   DATA[2227,0] := 2.649009;
   DATA[2227,1] := 864.9738;
   DATA[2227,2] := 2.0;
   DATA[2227,3] := 2.0;
   DATA[2227,4] := 262.3366;
   DATA[2227,5] := 8.394514;
   DATA[2227,6] := 330.2999;
   DATA[2227,7] := 2.461539;
   DATA[2227,8] := 2.0;
   DATA[2227,9] := 2.0;
   DATA[2227,10] := 2.0;
   DATA[2227,11] := 19.73878;
   DATA[2227,12] := 2.209653;
   DATA[2227,13] := 811.05;
   DATA[2227,14] := 1.0;
   DATA[2227,15] := 2.0;
   DATA[2227,16] := 1.0;
   DATA[2227,17] := 1.0;
   DATA[2227,18] := 1.0;
   DATA[2227,19] := 2.0;
   DATA[2227,20] := 148.808;
   DATA[2227,21] := 155.0884;
   DATA[2227,22] := 1.715567;
   DATA[2227,23] := 847.5134;
   DATA[2227,24] := 2.0;
   DATA[2227,25] := 2.0;
   DATA[2227,26] := 7.873815;
   DATA[2227,27] := 144.2194;
   DATA[2227,28] := 261.8559;
   DATA[2227,29] := 11.88157;
   DATA[2227,30] := 1.726865;
   DATA[2227,31] := 1.281927;
   DATA[2227,32] := 0.7352687;
   DATA[2227,33] := 0.3084905;
   DATA[2227,34] := 2.0;
   DATA[2227,35] := 250.016;
   DATA[2227,36] := 1.69801;
   DATA[2227,37] := 188.9259;
   DATA[2227,38] := 0.000128152;
   DATA[2227,39] := 1.0;
   DATA[2227,40] := 1.0;
   DATA[2228,0] := 2.653813;
   DATA[2228,1] := 865.013;
   DATA[2228,2] := 2.0;
   DATA[2228,3] := 2.0;
   DATA[2228,4] := 262.3366;
   DATA[2228,5] := 8.394514;
   DATA[2228,6] := 330.2999;
   DATA[2228,7] := 2.461539;
   DATA[2228,8] := 2.0;
   DATA[2228,9] := 2.0;
   DATA[2228,10] := 2.0;
   DATA[2228,11] := 19.73878;
   DATA[2228,12] := 2.209653;
   DATA[2228,13] := 811.01;
   DATA[2228,14] := 1.0;
   DATA[2228,15] := 2.0;
   DATA[2228,16] := 1.0;
   DATA[2228,17] := 1.0;
   DATA[2228,18] := 1.0;
   DATA[2228,19] := 2.0;
   DATA[2228,20] := 148.808;
   DATA[2228,21] := 155.0884;
   DATA[2228,22] := 1.715567;
   DATA[2228,23] := 847.5903;
   DATA[2228,24] := 2.0;
   DATA[2228,25] := 2.0;
   DATA[2228,26] := 7.873815;
   DATA[2228,27] := 144.2194;
   DATA[2228,28] := 261.8559;
   DATA[2228,29] := 11.88157;
   DATA[2228,30] := 1.726865;
   DATA[2228,31] := 1.281927;
   DATA[2228,32] := 0.7352687;
   DATA[2228,33] := 0.3084905;
   DATA[2228,34] := 2.0;
   DATA[2228,35] := 249.9359;
   DATA[2228,36] := 1.69801;
   DATA[2228,37] := 188.9259;
   DATA[2228,38] := 0.000128152;
   DATA[2228,39] := 1.0;
   DATA[2228,40] := 1.0;
   DATA[2229,0] := 2.643564;
   DATA[2229,1] := 864.8168;
   DATA[2229,2] := 2.0;
   DATA[2229,3] := 2.0;
   DATA[2229,4] := 262.3366;
   DATA[2229,5] := 8.394514;
   DATA[2229,6] := 330.2999;
   DATA[2229,7] := 2.460129;
   DATA[2229,8] := 2.0;
   DATA[2229,9] := 2.0;
   DATA[2229,10] := 2.0;
   DATA[2229,11] := 19.82201;
   DATA[2229,12] := 2.207603;
   DATA[2229,13] := 811.01;
   DATA[2229,14] := 1.0;
   DATA[2229,15] := 2.0;
   DATA[2229,16] := 1.0;
   DATA[2229,17] := 1.0;
   DATA[2229,18] := 1.0;
   DATA[2229,19] := 2.0;
   DATA[2229,20] := 148.808;
   DATA[2229,21] := 155.0884;
   DATA[2229,22] := 1.716849;
   DATA[2229,23] := 847.6288;
   DATA[2229,24] := 2.0;
   DATA[2229,25] := 2.0;
   DATA[2229,26] := 7.873815;
   DATA[2229,27] := 144.2194;
   DATA[2229,28] := 261.8559;
   DATA[2229,29] := 12.11228;
   DATA[2229,30] := 1.726865;
   DATA[2229,31] := 1.281927;
   DATA[2229,32] := 0.7352687;
   DATA[2229,33] := 0.3084905;
   DATA[2229,34] := 2.0;
   DATA[2229,35] := 249.9359;
   DATA[2229,36] := 1.69801;
   DATA[2229,37] := 188.9259;
   DATA[2229,38] := 0.000128152;
   DATA[2229,39] := 1.0;
   DATA[2229,40] := 1.0;
   DATA[2230,0] := 2.624988;
   DATA[2230,1] := 864.9738;
   DATA[2230,2] := 2.0;
   DATA[2230,3] := 2.0;
   DATA[2230,4] := 262.3366;
   DATA[2230,5] := 8.394514;
   DATA[2230,6] := 330.2999;
   DATA[2230,7] := 2.458206;
   DATA[2230,8] := 2.0;
   DATA[2230,9] := 2.0;
   DATA[2230,10] := 2.0;
   DATA[2230,11] := 19.82201;
   DATA[2230,12] := 2.207347;
   DATA[2230,13] := 810.9299;
   DATA[2230,14] := 1.0;
   DATA[2230,15] := 2.0;
   DATA[2230,16] := 1.0;
   DATA[2230,17] := 1.0;
   DATA[2230,18] := 1.0;
   DATA[2230,19] := 2.0;
   DATA[2230,20] := 148.808;
   DATA[2230,21] := 155.0884;
   DATA[2230,22] := 1.717361;
   DATA[2230,23] := 847.7057;
   DATA[2230,24] := 2.0;
   DATA[2230,25] := 2.0;
   DATA[2230,26] := 7.873815;
   DATA[2230,27] := 144.2194;
   DATA[2230,28] := 261.8559;
   DATA[2230,29] := 12.11228;
   DATA[2230,30] := 1.726865;
   DATA[2230,31] := 1.281927;
   DATA[2230,32] := 0.7352687;
   DATA[2230,33] := 0.3084905;
   DATA[2230,34] := 2.0;
   DATA[2230,35] := 249.9359;
   DATA[2230,36] := 1.69801;
   DATA[2230,37] := 188.9259;
   DATA[2230,38] := 0.000128152;
   DATA[2230,39] := 1.0;
   DATA[2230,40] := 1.0;
   DATA[2231,0] := 2.620504;
   DATA[2231,1] := 865.013;
   DATA[2231,2] := 2.0;
   DATA[2231,3] := 2.0;
   DATA[2231,4] := 262.3366;
   DATA[2231,5] := 8.394514;
   DATA[2231,6] := 330.2999;
   DATA[2231,7] := 2.458078;
   DATA[2231,8] := 2.0;
   DATA[2231,9] := 2.0;
   DATA[2231,10] := 2.0;
   DATA[2231,11] := 19.82201;
   DATA[2231,12] := 2.207347;
   DATA[2231,13] := 810.8498;
   DATA[2231,14] := 1.0;
   DATA[2231,15] := 2.0;
   DATA[2231,16] := 1.0;
   DATA[2231,17] := 1.0;
   DATA[2231,18] := 1.0;
   DATA[2231,19] := 2.0;
   DATA[2231,20] := 148.808;
   DATA[2231,21] := 155.0884;
   DATA[2231,22] := 1.717361;
   DATA[2231,23] := 847.821;
   DATA[2231,24] := 2.0;
   DATA[2231,25] := 2.0;
   DATA[2231,26] := 7.873815;
   DATA[2231,27] := 144.2194;
   DATA[2231,28] := 261.8559;
   DATA[2231,29] := 12.11228;
   DATA[2231,30] := 1.728531;
   DATA[2231,31] := 1.281927;
   DATA[2231,32] := 0.7352687;
   DATA[2231,33] := 0.3084905;
   DATA[2231,34] := 2.0;
   DATA[2231,35] := 249.9359;
   DATA[2231,36] := 1.69801;
   DATA[2231,37] := 188.9259;
   DATA[2231,38] := 0.000128152;
   DATA[2231,39] := 1.0;
   DATA[2231,40] := 1.0;
   DATA[2232,0] := 2.616981;
   DATA[2232,1] := 865.013;
   DATA[2232,2] := 2.0;
   DATA[2232,3] := 2.0;
   DATA[2232,4] := 262.3366;
   DATA[2232,5] := 8.394514;
   DATA[2232,6] := 330.2999;
   DATA[2232,7] := 2.455772;
   DATA[2232,8] := 2.0;
   DATA[2232,9] := 2.0;
   DATA[2232,10] := 2.0;
   DATA[2232,11] := 19.74198;
   DATA[2232,12] := 2.207347;
   DATA[2232,13] := 811.1302;
   DATA[2232,14] := 1.0;
   DATA[2232,15] := 2.0;
   DATA[2232,16] := 1.0;
   DATA[2232,17] := 1.0;
   DATA[2232,18] := 1.0;
   DATA[2232,19] := 2.0;
   DATA[2232,20] := 148.808;
   DATA[2232,21] := 155.0884;
   DATA[2232,22] := 1.717361;
   DATA[2232,23] := 847.6288;
   DATA[2232,24] := 2.0;
   DATA[2232,25] := 2.0;
   DATA[2232,26] := 7.873815;
   DATA[2232,27] := 144.2194;
   DATA[2232,28] := 261.8559;
   DATA[2232,29] := 12.11228;
   DATA[2232,30] := 1.728659;
   DATA[2232,31] := 1.268989;
   DATA[2232,32] := 0.7352687;
   DATA[2232,33] := 0.3084905;
   DATA[2232,34] := 2.0;
   DATA[2232,35] := 250.1122;
   DATA[2232,36] := 1.69801;
   DATA[2232,37] := 188.9259;
   DATA[2232,38] := 0.000128152;
   DATA[2232,39] := 1.0;
   DATA[2232,40] := 1.0;
   DATA[2233,0] := 2.609615;
   DATA[2233,1] := 865.2485;
   DATA[2233,2] := 2.0;
   DATA[2233,3] := 2.0;
   DATA[2233,4] := 262.3366;
   DATA[2233,5] := 8.396757;
   DATA[2233,6] := 330.2999;
   DATA[2233,7] := 2.456412;
   DATA[2233,8] := 2.0;
   DATA[2233,9] := 2.0;
   DATA[2233,10] := 2.0;
   DATA[2233,11] := 19.71957;
   DATA[2233,12] := 2.207347;
   DATA[2233,13] := 811.1302;
   DATA[2233,14] := 1.0;
   DATA[2233,15] := 2.0;
   DATA[2233,16] := 1.0;
   DATA[2233,17] := 1.0;
   DATA[2233,18] := 1.0;
   DATA[2233,19] := 2.0;
   DATA[2233,20] := 148.808;
   DATA[2233,21] := 155.0884;
   DATA[2233,22] := 1.717361;
   DATA[2233,23] := 847.821;
   DATA[2233,24] := 2.0;
   DATA[2233,25] := 2.0;
   DATA[2233,26] := 7.873815;
   DATA[2233,27] := 144.2194;
   DATA[2233,28] := 261.8559;
   DATA[2233,29] := 12.11228;
   DATA[2233,30] := 1.728659;
   DATA[2233,31] := 1.261816;
   DATA[2233,32] := 0.7352687;
   DATA[2233,33] := 0.3084905;
   DATA[2233,34] := 2.0;
   DATA[2233,35] := 250.2243;
   DATA[2233,36] := 1.69801;
   DATA[2233,37] := 188.9259;
   DATA[2233,38] := 0.000128152;
   DATA[2233,39] := 1.0;
   DATA[2233,40] := 1.0;
   DATA[2234,0] := 2.588156;
   DATA[2234,1] := 865.013;
   DATA[2234,2] := 2.0;
   DATA[2234,3] := 2.0;
   DATA[2234,4] := 262.3366;
   DATA[2234,5] := 8.396757;
   DATA[2234,6] := 330.2999;
   DATA[2234,7] := 2.458078;
   DATA[2234,8] := 2.0;
   DATA[2234,9] := 2.0;
   DATA[2234,10] := 2.0;
   DATA[2234,11] := 19.71957;
   DATA[2234,12] := 2.206963;
   DATA[2234,13] := 811.05;
   DATA[2234,14] := 1.0;
   DATA[2234,15] := 2.0;
   DATA[2234,16] := 1.0;
   DATA[2234,17] := 1.0;
   DATA[2234,18] := 1.0;
   DATA[2234,19] := 2.0;
   DATA[2234,20] := 148.808;
   DATA[2234,21] := 155.0884;
   DATA[2234,22] := 1.717361;
   DATA[2234,23] := 847.8979;
   DATA[2234,24] := 2.0;
   DATA[2234,25] := 2.0;
   DATA[2234,26] := 7.873815;
   DATA[2234,27] := 144.2194;
   DATA[2234,28] := 261.8559;
   DATA[2234,29] := 11.88157;
   DATA[2234,30] := 1.728659;
   DATA[2234,31] := 1.261816;
   DATA[2234,32] := 0.7352687;
   DATA[2234,33] := 0.3082983;
   DATA[2234,34] := 2.0;
   DATA[2234,35] := 250.2243;
   DATA[2234,36] := 1.69801;
   DATA[2234,37] := 188.974;
   DATA[2234,38] := 0.000128152;
   DATA[2234,39] := 1.0;
   DATA[2234,40] := 1.0;
   DATA[2235,0] := 2.5699;
   DATA[2235,1] := 864.9345;
   DATA[2235,2] := 2.0;
   DATA[2235,3] := 2.0;
   DATA[2235,4] := 262.3366;
   DATA[2235,5] := 8.396757;
   DATA[2235,6] := 330.2999;
   DATA[2235,7] := 2.458078;
   DATA[2235,8] := 2.0;
   DATA[2235,9] := 2.0;
   DATA[2235,10] := 2.0;
   DATA[2235,11] := 19.71957;
   DATA[2235,12] := 2.206963;
   DATA[2235,13] := 811.01;
   DATA[2235,14] := 1.0;
   DATA[2235,15] := 2.0;
   DATA[2235,16] := 1.0;
   DATA[2235,17] := 1.0;
   DATA[2235,18] := 1.0;
   DATA[2235,19] := 2.0;
   DATA[2235,20] := 148.808;
   DATA[2235,21] := 155.0372;
   DATA[2235,22] := 1.717361;
   DATA[2235,23] := 847.9364;
   DATA[2235,24] := 2.0;
   DATA[2235,25] := 2.0;
   DATA[2235,26] := 7.873815;
   DATA[2235,27] := 144.2194;
   DATA[2235,28] := 261.8559;
   DATA[2235,29] := 11.88157;
   DATA[2235,30] := 1.728659;
   DATA[2235,31] := 1.276419;
   DATA[2235,32] := 0.7352687;
   DATA[2235,33] := 0.3074016;
   DATA[2235,34] := 2.0;
   DATA[2235,35] := 250.2243;
   DATA[2235,36] := 1.69801;
   DATA[2235,37] := 189.1182;
   DATA[2235,38] := 0.000128152;
   DATA[2235,39] := 1.0;
   DATA[2235,40] := 1.0;
   DATA[2236,0] := 2.554847;
   DATA[2236,1] := 864.8168;
   DATA[2236,2] := 2.0;
   DATA[2236,3] := 2.0;
   DATA[2236,4] := 262.3366;
   DATA[2236,5] := 8.396757;
   DATA[2236,6] := 330.2999;
   DATA[2236,7] := 2.458078;
   DATA[2236,8] := 2.0;
   DATA[2236,9] := 2.0;
   DATA[2236,10] := 2.0;
   DATA[2236,11] := 19.71957;
   DATA[2236,12] := 2.206963;
   DATA[2236,13] := 811.05;
   DATA[2236,14] := 1.0;
   DATA[2236,15] := 2.0;
   DATA[2236,16] := 1.0;
   DATA[2236,17] := 1.0;
   DATA[2236,18] := 1.0;
   DATA[2236,19] := 2.0;
   DATA[2236,20] := 148.808;
   DATA[2236,21] := 155.0372;
   DATA[2236,22] := 1.718771;
   DATA[2236,23] := 847.821;
   DATA[2236,24] := 2.0;
   DATA[2236,25] := 2.0;
   DATA[2236,26] := 7.873815;
   DATA[2236,27] := 144.2194;
   DATA[2236,28] := 261.8559;
   DATA[2236,29] := 11.88157;
   DATA[2236,30] := 1.728659;
   DATA[2236,31] := 1.282311;
   DATA[2236,32] := 0.7352687;
   DATA[2236,33] := 0.306761;
   DATA[2236,34] := 2.0;
   DATA[2236,35] := 250.3365;
   DATA[2236,36] := 1.69801;
   DATA[2236,37] := 189.1182;
   DATA[2236,38] := 0.000128152;
   DATA[2236,39] := 1.0;
   DATA[2236,40] := 1.0;
   DATA[2237,0] := 2.53467;
   DATA[2237,1] := 864.4243;
   DATA[2237,2] := 2.0;
   DATA[2237,3] := 2.0;
   DATA[2237,4] := 262.3366;
   DATA[2237,5] := 8.396757;
   DATA[2237,6] := 330.2999;
   DATA[2237,7] := 2.457438;
   DATA[2237,8] := 2.0;
   DATA[2237,9] := 2.0;
   DATA[2237,10] := 2.0;
   DATA[2237,11] := 19.72598;
   DATA[2237,12] := 2.209653;
   DATA[2237,13] := 810.6495;
   DATA[2237,14] := 1.0;
   DATA[2237,15] := 2.0;
   DATA[2237,16] := 1.0;
   DATA[2237,17] := 1.0;
   DATA[2237,18] := 1.0;
   DATA[2237,19] := 2.0;
   DATA[2237,20] := 148.808;
   DATA[2237,21] := 155.0372;
   DATA[2237,22] := 1.718771;
   DATA[2237,23] := 847.9364;
   DATA[2237,24] := 2.0;
   DATA[2237,25] := 2.0;
   DATA[2237,26] := 7.873815;
   DATA[2237,27] := 144.2194;
   DATA[2237,28] := 261.8559;
   DATA[2237,29] := 11.88157;
   DATA[2237,30] := 1.728659;
   DATA[2237,31] := 1.26758;
   DATA[2237,32] := 0.7352687;
   DATA[2237,33] := 0.306761;
   DATA[2237,34] := 2.0;
   DATA[2237,35] := 250.3365;
   DATA[2237,36] := 1.69801;
   DATA[2237,37] := 189.1182;
   DATA[2237,38] := 0.000128152;
   DATA[2237,39] := 1.0;
   DATA[2237,40] := 1.0;
   DATA[2238,0] := 2.516734;
   DATA[2238,1] := 864.1887;
   DATA[2238,2] := 2.0;
   DATA[2238,3] := 2.0;
   DATA[2238,4] := 262.3366;
   DATA[2238,5] := 8.396757;
   DATA[2238,6] := 330.2999;
   DATA[2238,7] := 2.456541;
   DATA[2238,8] := 2.0;
   DATA[2238,9] := 2.0;
   DATA[2238,10] := 2.0;
   DATA[2238,11] := 19.72598;
   DATA[2238,12] := 2.209653;
   DATA[2238,13] := 810.8498;
   DATA[2238,14] := 1.0;
   DATA[2238,15] := 2.0;
   DATA[2238,16] := 1.0;
   DATA[2238,17] := 1.0;
   DATA[2238,18] := 1.0;
   DATA[2238,19] := 2.0;
   DATA[2238,20] := 148.808;
   DATA[2238,21] := 155.0372;
   DATA[2238,22] := 1.718771;
   DATA[2238,23] := 848.2056;
   DATA[2238,24] := 2.0;
   DATA[2238,25] := 2.0;
   DATA[2238,26] := 7.873815;
   DATA[2238,27] := 144.2194;
   DATA[2238,28] := 261.8559;
   DATA[2238,29] := 11.88157;
   DATA[2238,30] := 1.727378;
   DATA[2238,31] := 1.256821;
   DATA[2238,32] := 0.7352687;
   DATA[2238,33] := 0.306761;
   DATA[2238,34] := 2.0;
   DATA[2238,35] := 250.4646;
   DATA[2238,36] := 1.69801;
   DATA[2238,37] := 189.1182;
   DATA[2238,38] := 0.000128152;
   DATA[2238,39] := 1.0;
   DATA[2238,40] := 1.0;
   DATA[2239,0] := 2.498479;
   DATA[2239,1] := 864.3457;
   DATA[2239,2] := 2.0;
   DATA[2239,3] := 2.0;
   DATA[2239,4] := 262.3366;
   DATA[2239,5] := 8.394835;
   DATA[2239,6] := 330.2999;
   DATA[2239,7] := 2.456541;
   DATA[2239,8] := 2.0;
   DATA[2239,9] := 2.0;
   DATA[2239,10] := 2.0;
   DATA[2239,11] := 19.75799;
   DATA[2239,12] := 2.208244;
   DATA[2239,13] := 810.5694;
   DATA[2239,14] := 1.0;
   DATA[2239,15] := 2.0;
   DATA[2239,16] := 1.0;
   DATA[2239,17] := 1.0;
   DATA[2239,18] := 1.0;
   DATA[2239,19] := 2.0;
   DATA[2239,20] := 148.808;
   DATA[2239,21] := 155.0372;
   DATA[2239,22] := 1.718771;
   DATA[2239,23] := 848.1671;
   DATA[2239,24] := 2.0;
   DATA[2239,25] := 2.0;
   DATA[2239,26] := 7.873815;
   DATA[2239,27] := 144.2194;
   DATA[2239,28] := 261.8559;
   DATA[2239,29] := 12.03538;
   DATA[2239,30] := 1.725968;
   DATA[2239,31] := 1.254259;
   DATA[2239,32] := 0.7352687;
   DATA[2239,33] := 0.306761;
   DATA[2239,34] := 2.0;
   DATA[2239,35] := 250.4646;
   DATA[2239,36] := 1.69801;
   DATA[2239,37] := 189.1182;
   DATA[2239,38] := 0.000128152;
   DATA[2239,39] := 1.0;
   DATA[2239,40] := 1.0;
   DATA[2240,0] := 2.484707;
   DATA[2240,1] := 863.9532;
   DATA[2240,2] := 2.0;
   DATA[2240,3] := 2.0;
   DATA[2240,4] := 262.3366;
   DATA[2240,5] := 8.394835;
   DATA[2240,6] := 330.2999;
   DATA[2240,7] := 2.456541;
   DATA[2240,8] := 2.0;
   DATA[2240,9] := 2.0;
   DATA[2240,10] := 2.0;
   DATA[2240,11] := 19.75799;
   DATA[2240,12] := 2.20645;
   DATA[2240,13] := 810.5294;
   DATA[2240,14] := 1.0;
   DATA[2240,15] := 2.0;
   DATA[2240,16] := 1.0;
   DATA[2240,17] := 1.0;
   DATA[2240,18] := 1.0;
   DATA[2240,19] := 2.0;
   DATA[2240,20] := 148.808;
   DATA[2240,21] := 155.0884;
   DATA[2240,22] := 1.717874;
   DATA[2240,23] := 848.3209;
   DATA[2240,24] := 2.0;
   DATA[2240,25] := 2.0;
   DATA[2240,26] := 7.873815;
   DATA[2240,27] := 144.2194;
   DATA[2240,28] := 261.7278;
   DATA[2240,29] := 12.15073;
   DATA[2240,30] := 1.724686;
   DATA[2240,31] := 1.254259;
   DATA[2240,32] := 0.7352687;
   DATA[2240,33] := 0.306761;
   DATA[2240,34] := 2.0;
   DATA[2240,35] := 250.4646;
   DATA[2240,36] := 1.69801;
   DATA[2240,37] := 189.1182;
   DATA[2240,38] := 0.000128152;
   DATA[2240,39] := 1.0;
   DATA[2240,40] := 1.0;
   DATA[2241,0] := 2.472216;
   DATA[2241,1] := 863.2859;
   DATA[2241,2] := 2.0;
   DATA[2241,3] := 2.0;
   DATA[2241,4] := 262.3366;
   DATA[2241,5] := 8.394835;
   DATA[2241,6] := 330.2999;
   DATA[2241,7] := 2.455643;
   DATA[2241,8] := 2.0;
   DATA[2241,9] := 2.0;
   DATA[2241,10] := 2.0;
   DATA[2241,11] := 19.73238;
   DATA[2241,12] := 2.20645;
   DATA[2241,13] := 810.4493;
   DATA[2241,14] := 1.0;
   DATA[2241,15] := 2.0;
   DATA[2241,16] := 1.0;
   DATA[2241,17] := 1.0;
   DATA[2241,18] := 1.0;
   DATA[2241,19] := 2.0;
   DATA[2241,20] := 148.808;
   DATA[2241,21] := 155.191;
   DATA[2241,22] := 1.717489;
   DATA[2241,23] := 848.3978;
   DATA[2241,24] := 2.0;
   DATA[2241,25] := 2.0;
   DATA[2241,26] := 7.873815;
   DATA[2241,27] := 144.2194;
   DATA[2241,28] := 261.7278;
   DATA[2241,29] := 12.15073;
   DATA[2241,30] := 1.724686;
   DATA[2241,31] := 1.270783;
   DATA[2241,32] := 0.7352687;
   DATA[2241,33] := 0.306761;
   DATA[2241,34] := 2.0;
   DATA[2241,35] := 250.3365;
   DATA[2241,36] := 1.69801;
   DATA[2241,37] := 189.1182;
   DATA[2241,38] := 0.000128152;
   DATA[2241,39] := 1.0;
   DATA[2241,40] := 1.0;
   DATA[2242,0] := 2.460366;
   DATA[2242,1] := 863.0897;
   DATA[2242,2] := 2.0;
   DATA[2242,3] := 2.0;
   DATA[2242,4] := 262.3366;
   DATA[2242,5] := 8.394835;
   DATA[2242,6] := 330.2999;
   DATA[2242,7] := 2.455643;
   DATA[2242,8] := 2.0;
   DATA[2242,9] := 2.0;
   DATA[2242,10] := 2.0;
   DATA[2242,11] := 19.70037;
   DATA[2242,12] := 2.20645;
   DATA[2242,13] := 810.249;
   DATA[2242,14] := 1.0;
   DATA[2242,15] := 2.0;
   DATA[2242,16] := 1.0;
   DATA[2242,17] := 1.0;
   DATA[2242,18] := 1.0;
   DATA[2242,19] := 2.0;
   DATA[2242,20] := 148.808;
   DATA[2242,21] := 155.191;
   DATA[2242,22] := 1.717489;
   DATA[2242,23] := 848.5516;
   DATA[2242,24] := 2.0;
   DATA[2242,25] := 2.0;
   DATA[2242,26] := 7.873815;
   DATA[2242,27] := 144.2451;
   DATA[2242,28] := 261.7278;
   DATA[2242,29] := 12.15073;
   DATA[2242,30] := 1.724686;
   DATA[2242,31] := 1.272064;
   DATA[2242,32] := 0.7352687;
   DATA[2242,33] := 0.3075297;
   DATA[2242,34] := 2.0;
   DATA[2242,35] := 250.2403;
   DATA[2242,36] := 1.69801;
   DATA[2242,37] := 189.1182;
   DATA[2242,38] := 0.000128152;
   DATA[2242,39] := 1.0;
   DATA[2242,40] := 1.0;
   DATA[2243,0] := 2.445633;
   DATA[2243,1] := 863.0897;
   DATA[2243,2] := 2.0;
   DATA[2243,3] := 2.0;
   DATA[2243,4] := 262.3366;
   DATA[2243,5] := 8.394835;
   DATA[2243,6] := 330.2999;
   DATA[2243,7] := 2.455643;
   DATA[2243,8] := 2.0;
   DATA[2243,9] := 2.0;
   DATA[2243,10] := 2.0;
   DATA[2243,11] := 19.70037;
   DATA[2243,12] := 2.20645;
   DATA[2243,13] := 810.3291;
   DATA[2243,14] := 1.0;
   DATA[2243,15] := 2.0;
   DATA[2243,16] := 1.0;
   DATA[2243,17] := 1.0;
   DATA[2243,18] := 1.0;
   DATA[2243,19] := 2.0;
   DATA[2243,20] := 148.808;
   DATA[2243,21] := 155.191;
   DATA[2243,22] := 1.717489;
   DATA[2243,23] := 847.9364;
   DATA[2243,24] := 2.0;
   DATA[2243,25] := 2.0;
   DATA[2243,26] := 7.873815;
   DATA[2243,27] := 144.2451;
   DATA[2243,28] := 261.7278;
   DATA[2243,29] := 12.15073;
   DATA[2243,30] := 1.724686;
   DATA[2243,31] := 1.272064;
   DATA[2243,32] := 0.7352687;
   DATA[2243,33] := 0.3079781;
   DATA[2243,34] := 2.0;
   DATA[2243,35] := 250.2403;
   DATA[2243,36] := 1.69801;
   DATA[2243,37] := 189.1182;
   DATA[2243,38] := 0.000128152;
   DATA[2243,39] := 1.0;
   DATA[2243,40] := 1.0;
   DATA[2244,0] := 2.435064;
   DATA[2244,1] := 862.8934;
   DATA[2244,2] := 2.0;
   DATA[2244,3] := 2.0;
   DATA[2244,4] := 262.3366;
   DATA[2244,5] := 8.394835;
   DATA[2244,6] := 330.2999;
   DATA[2244,7] := 2.455643;
   DATA[2244,8] := 2.0;
   DATA[2244,9] := 2.0;
   DATA[2244,10] := 2.0;
   DATA[2244,11] := 19.70037;
   DATA[2244,12] := 2.20645;
   DATA[2244,13] := 810.1689;
   DATA[2244,14] := 1.0;
   DATA[2244,15] := 2.0;
   DATA[2244,16] := 1.0;
   DATA[2244,17] := 1.0;
   DATA[2244,18] := 1.0;
   DATA[2244,19] := 2.0;
   DATA[2244,20] := 148.808;
   DATA[2244,21] := 155.191;
   DATA[2244,22] := 1.716464;
   DATA[2244,23] := 847.9364;
   DATA[2244,24] := 2.0;
   DATA[2244,25] := 2.0;
   DATA[2244,26] := 7.873815;
   DATA[2244,27] := 144.2451;
   DATA[2244,28] := 261.7278;
   DATA[2244,29] := 12.15073;
   DATA[2244,30] := 1.723789;
   DATA[2244,31] := 1.272064;
   DATA[2244,32] := 0.7352687;
   DATA[2244,33] := 0.3082983;
   DATA[2244,34] := 2.0;
   DATA[2244,35] := 250.2243;
   DATA[2244,36] := 1.69801;
   DATA[2244,37] := 189.006;
   DATA[2244,38] := 0.000128152;
   DATA[2244,39] := 1.0;
   DATA[2244,40] := 1.0;
   DATA[2245,0] := 2.428658;
   DATA[2245,1] := 862.8934;
   DATA[2245,2] := 2.0;
   DATA[2245,3] := 2.0;
   DATA[2245,4] := 262.3366;
   DATA[2245,5] := 8.394835;
   DATA[2245,6] := 330.2999;
   DATA[2245,7] := 2.458078;
   DATA[2245,8] := 2.0;
   DATA[2245,9] := 2.0;
   DATA[2245,10] := 2.0;
   DATA[2245,11] := 19.70037;
   DATA[2245,12] := 2.20645;
   DATA[2245,13] := 810.7296;
   DATA[2245,14] := 1.0;
   DATA[2245,15] := 2.0;
   DATA[2245,16] := 1.0;
   DATA[2245,17] := 1.0;
   DATA[2245,18] := 1.0;
   DATA[2245,19] := 2.0;
   DATA[2245,20] := 148.808;
   DATA[2245,21] := 155.191;
   DATA[2245,22] := 1.715567;
   DATA[2245,23] := 847.6288;
   DATA[2245,24] := 2.0;
   DATA[2245,25] := 2.0;
   DATA[2245,26] := 7.873815;
   DATA[2245,27] := 144.2451;
   DATA[2245,28] := 261.7278;
   DATA[2245,29] := 12.15073;
   DATA[2245,30] := 1.723789;
   DATA[2245,31] := 1.272064;
   DATA[2245,32] := 0.7352687;
   DATA[2245,33] := 0.3082983;
   DATA[2245,34] := 2.0;
   DATA[2245,35] := 250.1602;
   DATA[2245,36] := 1.69801;
   DATA[2245,37] := 188.8618;
   DATA[2245,38] := 0.000128152;
   DATA[2245,39] := 1.0;
   DATA[2245,40] := 1.0;
   DATA[2246,0] := 2.428658;
   DATA[2246,1] := 863.1682;
   DATA[2246,2] := 2.0;
   DATA[2246,3] := 2.0;
   DATA[2246,4] := 262.3366;
   DATA[2246,5] := 8.394835;
   DATA[2246,6] := 330.2999;
   DATA[2246,7] := 2.458078;
   DATA[2246,8] := 2.0;
   DATA[2246,9] := 2.0;
   DATA[2246,10] := 2.0;
   DATA[2246,11] := 19.70037;
   DATA[2246,12] := 2.20645;
   DATA[2246,13] := 810.5294;
   DATA[2246,14] := 1.0;
   DATA[2246,15] := 2.0;
   DATA[2246,16] := 1.0;
   DATA[2246,17] := 1.0;
   DATA[2246,18] := 1.0;
   DATA[2246,19] := 2.0;
   DATA[2246,20] := 148.808;
   DATA[2246,21] := 155.191;
   DATA[2246,22] := 1.715567;
   DATA[2246,23] := 847.7057;
   DATA[2246,24] := 2.0;
   DATA[2246,25] := 2.0;
   DATA[2246,26] := 7.873815;
   DATA[2246,27] := 144.2451;
   DATA[2246,28] := 261.7278;
   DATA[2246,29] := 12.15073;
   DATA[2246,30] := 1.725327;
   DATA[2246,31] := 1.278724;
   DATA[2246,32] := 0.7352687;
   DATA[2246,33] := 0.3082983;
   DATA[2246,34] := 2.0;
   DATA[2246,35] := 250.1602;
   DATA[2246,36] := 1.69801;
   DATA[2246,37] := 188.8618;
   DATA[2246,38] := 0.000128152;
   DATA[2246,39] := 1.0;
   DATA[2246,40] := 1.0;
   DATA[2247,0] := 2.451398;
   DATA[2247,1] := 863.1682;
   DATA[2247,2] := 2.0;
   DATA[2247,3] := 2.0;
   DATA[2247,4] := 262.3366;
   DATA[2247,5] := 8.394835;
   DATA[2247,6] := 330.2999;
   DATA[2247,7] := 2.458078;
   DATA[2247,8] := 2.0;
   DATA[2247,9] := 2.0;
   DATA[2247,10] := 2.0;
   DATA[2247,11] := 19.70037;
   DATA[2247,12] := 2.20645;
   DATA[2247,13] := 810.6495;
   DATA[2247,14] := 1.0;
   DATA[2247,15] := 2.0;
   DATA[2247,16] := 1.0;
   DATA[2247,17] := 1.0;
   DATA[2247,18] := 1.0;
   DATA[2247,19] := 2.0;
   DATA[2247,20] := 148.808;
   DATA[2247,21] := 155.191;
   DATA[2247,22] := 1.715567;
   DATA[2247,23] := 847.3212;
   DATA[2247,24] := 2.0;
   DATA[2247,25] := 2.0;
   DATA[2247,26] := 7.873815;
   DATA[2247,27] := 144.2451;
   DATA[2247,28] := 261.7278;
   DATA[2247,29] := 12.15073;
   DATA[2247,30] := 1.725327;
   DATA[2247,31] := 1.28167;
   DATA[2247,32] := 0.7352687;
   DATA[2247,33] := 0.3084905;
   DATA[2247,34] := 2.0;
   DATA[2247,35] := 250.1602;
   DATA[2247,36] := 1.69801;
   DATA[2247,37] := 188.8618;
   DATA[2247,38] := 0.000128152;
   DATA[2247,39] := 1.0;
   DATA[2247,40] := 1.0;
   DATA[2248,0] := 2.495916;
   DATA[2248,1] := 862.9719;
   DATA[2248,2] := 2.0;
   DATA[2248,3] := 2.0;
   DATA[2248,4] := 262.3366;
   DATA[2248,5] := 8.394835;
   DATA[2248,6] := 330.2999;
   DATA[2248,7] := 2.458078;
   DATA[2248,8] := 2.0;
   DATA[2248,9] := 2.0;
   DATA[2248,10] := 2.0;
   DATA[2248,11] := 19.64594;
   DATA[2248,12] := 2.20645;
   DATA[2248,13] := 810.7296;
   DATA[2248,14] := 1.0;
   DATA[2248,15] := 2.0;
   DATA[2248,16] := 1.0;
   DATA[2248,17] := 1.0;
   DATA[2248,18] := 1.0;
   DATA[2248,19] := 2.0;
   DATA[2248,20] := 148.808;
   DATA[2248,21] := 155.191;
   DATA[2248,22] := 1.715567;
   DATA[2248,23] := 847.3597;
   DATA[2248,24] := 2.0;
   DATA[2248,25] := 2.0;
   DATA[2248,26] := 7.873815;
   DATA[2248,27] := 144.2451;
   DATA[2248,28] := 261.7278;
   DATA[2248,29] := 12.15073;
   DATA[2248,30] := 1.725327;
   DATA[2248,31] := 1.282183;
   DATA[2248,32] := 0.7352687;
   DATA[2248,33] := 0.3084905;
   DATA[2248,34] := 2.0;
   DATA[2248,35] := 250.1602;
   DATA[2248,36] := 1.69801;
   DATA[2248,37] := 188.8618;
   DATA[2248,38] := 0.000128152;
   DATA[2248,39] := 1.0;
   DATA[2248,40] := 1.0;
   DATA[2249,0] := 2.541075;
   DATA[2249,1] := 863.3644;
   DATA[2249,2] := 2.0;
   DATA[2249,3] := 2.0;
   DATA[2249,4] := 262.3366;
   DATA[2249,5] := 8.394835;
   DATA[2249,6] := 330.2999;
   DATA[2249,7] := 2.458078;
   DATA[2249,8] := 2.0;
   DATA[2249,9] := 2.0;
   DATA[2249,10] := 2.0;
   DATA[2249,11] := 19.64594;
   DATA[2249,12] := 2.20645;
   DATA[2249,13] := 810.5294;
   DATA[2249,14] := 1.0;
   DATA[2249,15] := 2.0;
   DATA[2249,16] := 1.0;
   DATA[2249,17] := 1.0;
   DATA[2249,18] := 1.0;
   DATA[2249,19] := 2.0;
   DATA[2249,20] := 148.808;
   DATA[2249,21] := 155.191;
   DATA[2249,22] := 1.715567;
   DATA[2249,23] := 847.4366;
   DATA[2249,24] := 2.0;
   DATA[2249,25] := 2.0;
   DATA[2249,26] := 7.873815;
   DATA[2249,27] := 144.2451;
   DATA[2249,28] := 261.7278;
   DATA[2249,29] := 12.15073;
   DATA[2249,30] := 1.725327;
   DATA[2249,31] := 1.271423;
   DATA[2249,32] := 0.7352687;
   DATA[2249,33] := 0.3084905;
   DATA[2249,34] := 2.0;
   DATA[2249,35] := 250.1602;
   DATA[2249,36] := 1.601897;
   DATA[2249,37] := 188.8618;
   DATA[2249,38] := 0.000128152;
   DATA[2249,39] := 1.0;
   DATA[2249,40] := 1.0;
   DATA[2250,0] := 2.572463;
   DATA[2250,1] := 863.3644;
   DATA[2250,2] := 2.0;
   DATA[2250,3] := 2.0;
   DATA[2250,4] := 262.3366;
   DATA[2250,5] := 8.394835;
   DATA[2250,6] := 330.2999;
   DATA[2250,7] := 2.458078;
   DATA[2250,8] := 2.0;
   DATA[2250,9] := 2.0;
   DATA[2250,10] := 2.0;
   DATA[2250,11] := 19.74838;
   DATA[2250,12] := 2.20645;
   DATA[2250,13] := 811.01;
   DATA[2250,14] := 1.0;
   DATA[2250,15] := 2.0;
   DATA[2250,16] := 1.0;
   DATA[2250,17] := 1.0;
   DATA[2250,18] := 1.0;
   DATA[2250,19] := 2.0;
   DATA[2250,20] := 148.808;
   DATA[2250,21] := 155.191;
   DATA[2250,22] := 1.715567;
   DATA[2250,23] := 847.6288;
   DATA[2250,24] := 2.0;
   DATA[2250,25] := 2.0;
   DATA[2250,26] := 7.873815;
   DATA[2250,27] := 144.2451;
   DATA[2250,28] := 261.7278;
   DATA[2250,29] := 11.95847;
   DATA[2250,30] := 1.725327;
   DATA[2250,31] := 1.271423;
   DATA[2250,32] := 0.7352687;
   DATA[2250,33] := 0.3084905;
   DATA[2250,34] := 2.0;
   DATA[2250,35] := 250.1602;
   DATA[2250,36] := 1.601897;
   DATA[2250,37] := 188.8618;
   DATA[2250,38] := 0.000128152;
   DATA[2250,39] := 1.0;
   DATA[2250,40] := 1.0;
   DATA[2251,0] := 2.613138;
   DATA[2251,1] := 863.8354;
   DATA[2251,2] := 2.0;
   DATA[2251,3] := 2.0;
   DATA[2251,4] := 262.3366;
   DATA[2251,5] := 8.394835;
   DATA[2251,6] := 330.2999;
   DATA[2251,7] := 2.456797;
   DATA[2251,8] := 2.0;
   DATA[2251,9] := 2.0;
   DATA[2251,10] := 2.0;
   DATA[2251,11] := 19.75799;
   DATA[2251,12] := 2.208756;
   DATA[2251,13] := 810.5694;
   DATA[2251,14] := 1.0;
   DATA[2251,15] := 2.0;
   DATA[2251,16] := 1.0;
   DATA[2251,17] := 1.0;
   DATA[2251,18] := 1.0;
   DATA[2251,19] := 2.0;
   DATA[2251,20] := 148.808;
   DATA[2251,21] := 155.191;
   DATA[2251,22] := 1.715567;
   DATA[2251,23] := 847.7057;
   DATA[2251,24] := 2.0;
   DATA[2251,25] := 2.0;
   DATA[2251,26] := 7.873815;
   DATA[2251,27] := 144.2451;
   DATA[2251,28] := 261.7278;
   DATA[2251,29] := 11.95847;
   DATA[2251,30] := 1.725327;
   DATA[2251,31] := 1.271423;
   DATA[2251,32] := 0.7352687;
   DATA[2251,33] := 0.3084905;
   DATA[2251,34] := 2.0;
   DATA[2251,35] := 250.1602;
   DATA[2251,36] := 1.601897;
   DATA[2251,37] := 188.8618;
   DATA[2251,38] := 0.000128152;
   DATA[2251,39] := 1.0;
   DATA[2251,40] := 1.0;
   DATA[2252,0] := 2.630753;
   DATA[2252,1] := 863.9924;
   DATA[2252,2] := 2.0;
   DATA[2252,3] := 2.0;
   DATA[2252,4] := 262.3366;
   DATA[2252,5] := 8.394835;
   DATA[2252,6] := 330.2999;
   DATA[2252,7] := 2.456541;
   DATA[2252,8] := 2.0;
   DATA[2252,9] := 2.0;
   DATA[2252,10] := 2.0;
   DATA[2252,11] := 19.77079;
   DATA[2252,12] := 2.208884;
   DATA[2252,13] := 810.8098;
   DATA[2252,14] := 1.0;
   DATA[2252,15] := 2.0;
   DATA[2252,16] := 1.0;
   DATA[2252,17] := 1.0;
   DATA[2252,18] := 1.0;
   DATA[2252,19] := 2.0;
   DATA[2252,20] := 148.808;
   DATA[2252,21] := 155.191;
   DATA[2252,22] := 1.717233;
   DATA[2252,23] := 847.7057;
   DATA[2252,24] := 2.0;
   DATA[2252,25] := 2.0;
   DATA[2252,26] := 7.873815;
   DATA[2252,27] := 144.0656;
   DATA[2252,28] := 261.7278;
   DATA[2252,29] := 11.95847;
   DATA[2252,30] := 1.725327;
   DATA[2252,31] := 1.264506;
   DATA[2252,32] := 0.7352687;
   DATA[2252,33] := 0.3084905;
   DATA[2252,34] := 2.0;
   DATA[2252,35] := 250.1602;
   DATA[2252,36] := 1.601897;
   DATA[2252,37] := 188.9419;
   DATA[2252,38] := 0.000128152;
   DATA[2252,39] := 1.0;
   DATA[2252,40] := 1.0;
   DATA[2253,0] := 2.646767;
   DATA[2253,1] := 864.542;
   DATA[2253,2] := 2.0;
   DATA[2253,3] := 2.0;
   DATA[2253,4] := 262.3366;
   DATA[2253,5] := 8.394835;
   DATA[2253,6] := 330.2999;
   DATA[2253,7] := 2.456541;
   DATA[2253,8] := 2.0;
   DATA[2253,9] := 2.0;
   DATA[2253,10] := 2.0;
   DATA[2253,11] := 19.70357;
   DATA[2253,12] := 2.209909;
   DATA[2253,13] := 811.1302;
   DATA[2253,14] := 1.0;
   DATA[2253,15] := 2.0;
   DATA[2253,16] := 1.0;
   DATA[2253,17] := 1.0;
   DATA[2253,18] := 1.0;
   DATA[2253,19] := 2.0;
   DATA[2253,20] := 148.808;
   DATA[2253,21] := 155.191;
   DATA[2253,22] := 1.717489;
   DATA[2253,23] := 847.7826;
   DATA[2253,24] := 2.0;
   DATA[2253,25] := 2.0;
   DATA[2253,26] := 7.873815;
   DATA[2253,27] := 144.0656;
   DATA[2253,28] := 261.7278;
   DATA[2253,29] := 11.95847;
   DATA[2253,30] := 1.725327;
   DATA[2253,31] := 1.262713;
   DATA[2253,32] := 0.7352687;
   DATA[2253,33] := 0.3084905;
   DATA[2253,34] := 2.0;
   DATA[2253,35] := 250.1602;
   DATA[2253,36] := 1.601897;
   DATA[2253,37] := 189.006;
   DATA[2253,38] := 0.000128152;
   DATA[2253,39] := 1.0;
   DATA[2253,40] := 1.0;
   DATA[2254,0] := 2.649329;
   DATA[2254,1] := 864.6205;
   DATA[2254,2] := 2.0;
   DATA[2254,3] := 2.0;
   DATA[2254,4] := 262.3366;
   DATA[2254,5] := 8.394835;
   DATA[2254,6] := 330.2999;
   DATA[2254,7] := 2.457566;
   DATA[2254,8] := 2.0;
   DATA[2254,9] := 2.0;
   DATA[2254,10] := 2.0;
   DATA[2254,11] := 19.65235;
   DATA[2254,12] := 2.21055;
   DATA[2254,13] := 811.3304;
   DATA[2254,14] := 1.0;
   DATA[2254,15] := 2.0;
   DATA[2254,16] := 1.0;
   DATA[2254,17] := 1.0;
   DATA[2254,18] := 1.0;
   DATA[2254,19] := 2.0;
   DATA[2254,20] := 148.808;
   DATA[2254,21] := 155.191;
   DATA[2254,22] := 1.717489;
   DATA[2254,23] := 847.5903;
   DATA[2254,24] := 2.0;
   DATA[2254,25] := 2.0;
   DATA[2254,26] := 7.874455;
   DATA[2254,27] := 144.0656;
   DATA[2254,28] := 261.7278;
   DATA[2254,29] := 11.95847;
   DATA[2254,30] := 1.725327;
   DATA[2254,31] := 1.271551;
   DATA[2254,32] := 0.7352687;
   DATA[2254,33] := 0.3084905;
   DATA[2254,34] := 2.0;
   DATA[2254,35] := 250.1602;
   DATA[2254,36] := 1.681991;
   DATA[2254,37] := 189.006;
   DATA[2254,38] := 0.000128152;
   DATA[2254,39] := 1.0;
   DATA[2254,40] := 1.0;
   DATA[2255,0] := 2.646126;
   DATA[2255,1] := 864.8168;
   DATA[2255,2] := 2.0;
   DATA[2255,3] := 2.0;
   DATA[2255,4] := 262.3366;
   DATA[2255,5] := 8.394835;
   DATA[2255,6] := 330.2999;
   DATA[2255,7] := 2.457822;
   DATA[2255,8] := 2.0;
   DATA[2255,9] := 2.0;
   DATA[2255,10] := 2.0;
   DATA[2255,11] := 19.64594;
   DATA[2255,12] := 2.21055;
   DATA[2255,13] := 811.6509;
   DATA[2255,14] := 1.0;
   DATA[2255,15] := 2.0;
   DATA[2255,16] := 1.0;
   DATA[2255,17] := 1.0;
   DATA[2255,18] := 1.0;
   DATA[2255,19] := 2.0;
   DATA[2255,20] := 148.808;
   DATA[2255,21] := 155.191;
   DATA[2255,22] := 1.717489;
   DATA[2255,23] := 848.1287;
   DATA[2255,24] := 2.0;
   DATA[2255,25] := 2.0;
   DATA[2255,26] := 7.874455;
   DATA[2255,27] := 144.0656;
   DATA[2255,28] := 261.7278;
   DATA[2255,29] := 11.95847;
   DATA[2255,30] := 1.725327;
   DATA[2255,31] := 1.280902;
   DATA[2255,32] := 0.7352687;
   DATA[2255,33] := 0.3084905;
   DATA[2255,34] := 2.0;
   DATA[2255,35] := 250.1602;
   DATA[2255,36] := 1.681991;
   DATA[2255,37] := 189.006;
   DATA[2255,38] := 0.000128152;
   DATA[2255,39] := 1.0;
   DATA[2255,40] := 1.0;
   DATA[2256,0] := 2.622746;
   DATA[2256,1] := 864.9345;
   DATA[2256,2] := 2.0;
   DATA[2256,3] := 2.0;
   DATA[2256,4] := 262.3366;
   DATA[2256,5] := 8.394835;
   DATA[2256,6] := 330.2999;
   DATA[2256,7] := 2.456541;
   DATA[2256,8] := 2.0;
   DATA[2256,9] := 2.0;
   DATA[2256,10] := 2.0;
   DATA[2256,11] := 19.64594;
   DATA[2256,12] := 2.21055;
   DATA[2256,13] := 811.731;
   DATA[2256,14] := 1.0;
   DATA[2256,15] := 2.0;
   DATA[2256,16] := 1.0;
   DATA[2256,17] := 1.0;
   DATA[2256,18] := 1.0;
   DATA[2256,19] := 2.0;
   DATA[2256,20] := 148.808;
   DATA[2256,21] := 155.191;
   DATA[2256,22] := 1.717489;
   DATA[2256,23] := 848.0133;
   DATA[2256,24] := 2.0;
   DATA[2256,25] := 2.0;
   DATA[2256,26] := 7.874455;
   DATA[2256,27] := 144.0656;
   DATA[2256,28] := 261.7278;
   DATA[2256,29] := 11.95847;
   DATA[2256,30] := 1.725327;
   DATA[2256,31] := 1.295376;
   DATA[2256,32] := 0.7352687;
   DATA[2256,33] := 0.306761;
   DATA[2256,34] := 2.0;
   DATA[2256,35] := 250.1602;
   DATA[2256,36] := 1.681991;
   DATA[2256,37] := 189.006;
   DATA[2256,38] := 0.000128152;
   DATA[2256,39] := 1.0;
   DATA[2256,40] := 1.0;
   DATA[2257,0] := 2.622746;
   DATA[2257,1] := 864.9345;
   DATA[2257,2] := 2.0;
   DATA[2257,3] := 2.0;
   DATA[2257,4] := 262.3366;
   DATA[2257,5] := 8.394835;
   DATA[2257,6] := 330.2999;
   DATA[2257,7] := 2.456541;
   DATA[2257,8] := 2.0;
   DATA[2257,9] := 2.0;
   DATA[2257,10] := 2.0;
   DATA[2257,11] := 19.64594;
   DATA[2257,12] := 2.21055;
   DATA[2257,13] := 811.731;
   DATA[2257,14] := 1.0;
   DATA[2257,15] := 2.0;
   DATA[2257,16] := 1.0;
   DATA[2257,17] := 1.0;
   DATA[2257,18] := 1.0;
   DATA[2257,19] := 2.0;
   DATA[2257,20] := 148.808;
   DATA[2257,21] := 155.191;
   DATA[2257,22] := 1.717489;
   DATA[2257,23] := 848.0133;
   DATA[2257,24] := 2.0;
   DATA[2257,25] := 2.0;
   DATA[2257,26] := 7.874455;
   DATA[2257,27] := 144.0656;
   DATA[2257,28] := 261.7278;
   DATA[2257,29] := 11.95847;
   DATA[2257,30] := 1.725327;
   DATA[2257,31] := 1.295376;
   DATA[2257,32] := 0.7352687;
   DATA[2257,33] := 0.306761;
   DATA[2257,34] := 2.0;
   DATA[2257,35] := 250.1602;
   DATA[2257,36] := 1.681991;
   DATA[2257,37] := 189.006;
   DATA[2257,38] := 0.000128152;
   DATA[2257,39] := 1.0;
   DATA[2257,40] := 1.0;
   DATA[2258,0] := 2.618582;
   DATA[2258,1] := 864.7383;
   DATA[2258,2] := 2.0;
   DATA[2258,3] := 2.0;
   DATA[2258,4] := 262.3366;
   DATA[2258,5] := 8.394835;
   DATA[2258,6] := 330.2999;
   DATA[2258,7] := 2.455772;
   DATA[2258,8] := 2.0;
   DATA[2258,9] := 2.0;
   DATA[2258,10] := 2.0;
   DATA[2258,11] := 19.64594;
   DATA[2258,12] := 2.21055;
   DATA[2258,13] := 811.9313;
   DATA[2258,14] := 1.0;
   DATA[2258,15] := 2.0;
   DATA[2258,16] := 1.0;
   DATA[2258,17] := 1.0;
   DATA[2258,18] := 1.0;
   DATA[2258,19] := 2.0;
   DATA[2258,20] := 148.808;
   DATA[2258,21] := 155.191;
   DATA[2258,22] := 1.717489;
   DATA[2258,23] := 848.1287;
   DATA[2258,24] := 2.0;
   DATA[2258,25] := 2.0;
   DATA[2258,26] := 7.874455;
   DATA[2258,27] := 144.0656;
   DATA[2258,28] := 261.7278;
   DATA[2258,29] := 11.95847;
   DATA[2258,30] := 1.725327;
   DATA[2258,31] := 1.299475;
   DATA[2258,32] := 0.7352687;
   DATA[2258,33] := 0.306761;
   DATA[2258,34] := 2.0;
   DATA[2258,35] := 250.1602;
   DATA[2258,36] := 1.681991;
   DATA[2258,37] := 189.006;
   DATA[2258,38] := 0.000128152;
   DATA[2258,39] := 1.0;
   DATA[2258,40] := 1.0;
   DATA[2259,0] := 2.613138;
   DATA[2259,1] := 864.7383;
   DATA[2259,2] := 2.0;
   DATA[2259,3] := 2.0;
   DATA[2259,4] := 262.3366;
   DATA[2259,5] := 8.394835;
   DATA[2259,6] := 330.2999;
   DATA[2259,7] := 2.455003;
   DATA[2259,8] := 2.0;
   DATA[2259,9] := 2.0;
   DATA[2259,10] := 2.0;
   DATA[2259,11] := 19.64594;
   DATA[2259,12] := 2.21055;
   DATA[2259,13] := 811.8511;
   DATA[2259,14] := 1.0;
   DATA[2259,15] := 2.0;
   DATA[2259,16] := 1.0;
   DATA[2259,17] := 1.0;
   DATA[2259,18] := 1.0;
   DATA[2259,19] := 2.0;
   DATA[2259,20] := 148.808;
   DATA[2259,21] := 155.191;
   DATA[2259,22] := 1.718002;
   DATA[2259,23] := 847.9364;
   DATA[2259,24] := 2.0;
   DATA[2259,25] := 2.0;
   DATA[2259,26] := 7.874455;
   DATA[2259,27] := 144.0656;
   DATA[2259,28] := 261.7278;
   DATA[2259,29] := 11.95847;
   DATA[2259,30] := 1.728531;
   DATA[2259,31] := 1.292046;
   DATA[2259,32] := 0.7352687;
   DATA[2259,33] := 0.306761;
   DATA[2259,34] := 2.0;
   DATA[2259,35] := 250.1762;
   DATA[2259,36] := 1.681991;
   DATA[2259,37] := 189.006;
   DATA[2259,38] := 0.000128152;
   DATA[2259,39] := 1.0;
   DATA[2259,40] := 1.0;
   DATA[2260,0] := 2.60417;
   DATA[2260,1] := 864.7775;
   DATA[2260,2] := 2.0;
   DATA[2260,3] := 2.0;
   DATA[2260,4] := 262.3366;
   DATA[2260,5] := 8.394835;
   DATA[2260,6] := 330.2999;
   DATA[2260,7] := 2.455003;
   DATA[2260,8] := 2.0;
   DATA[2260,9] := 2.0;
   DATA[2260,10] := 2.0;
   DATA[2260,11] := 19.64594;
   DATA[2260,12] := 2.209653;
   DATA[2260,13] := 811.8111;
   DATA[2260,14] := 1.0;
   DATA[2260,15] := 2.0;
   DATA[2260,16] := 1.0;
   DATA[2260,17] := 1.0;
   DATA[2260,18] := 1.0;
   DATA[2260,19] := 2.0;
   DATA[2260,20] := 148.808;
   DATA[2260,21] := 155.191;
   DATA[2260,22] := 1.719027;
   DATA[2260,23] := 848.2825;
   DATA[2260,24] := 2.0;
   DATA[2260,25] := 2.0;
   DATA[2260,26] := 7.874455;
   DATA[2260,27] := 144.0656;
   DATA[2260,28] := 261.7278;
   DATA[2260,29] := 11.95847;
   DATA[2260,30] := 1.728531;
   DATA[2260,31] := 1.282311;
   DATA[2260,32] := 0.7352687;
   DATA[2260,33] := 0.306761;
   DATA[2260,34] := 2.0;
   DATA[2260,35] := 250.3044;
   DATA[2260,36] := 1.681991;
   DATA[2260,37] := 189.1182;
   DATA[2260,38] := 0.000128152;
   DATA[2260,39] := 1.0;
   DATA[2260,40] := 1.0;
   DATA[2261,0] := 2.586555;
   DATA[2261,1] := 864.9738;
   DATA[2261,2] := 2.0;
   DATA[2261,3] := 2.0;
   DATA[2261,4] := 262.3366;
   DATA[2261,5] := 8.394835;
   DATA[2261,6] := 330.2999;
   DATA[2261,7] := 2.455003;
   DATA[2261,8] := 2.0;
   DATA[2261,9] := 2.0;
   DATA[2261,10] := 2.0;
   DATA[2261,11] := 19.70357;
   DATA[2261,12] := 2.209653;
   DATA[2261,13] := 812.1716;
   DATA[2261,14] := 1.0;
   DATA[2261,15] := 2.0;
   DATA[2261,16] := 1.0;
   DATA[2261,17] := 1.0;
   DATA[2261,18] := 1.0;
   DATA[2261,19] := 2.0;
   DATA[2261,20] := 148.808;
   DATA[2261,21] := 155.191;
   DATA[2261,22] := 1.719027;
   DATA[2261,23] := 848.3978;
   DATA[2261,24] := 2.0;
   DATA[2261,25] := 2.0;
   DATA[2261,26] := 7.874455;
   DATA[2261,27] := 144.2194;
   DATA[2261,28] := 261.7278;
   DATA[2261,29] := 11.95847;
   DATA[2261,30] := 1.728531;
   DATA[2261,31] := 1.273345;
   DATA[2261,32] := 0.7352687;
   DATA[2261,33] := 0.306761;
   DATA[2261,34] := 2.0;
   DATA[2261,35] := 250.3044;
   DATA[2261,36] := 1.681991;
   DATA[2261,37] := 189.1182;
   DATA[2261,38] := 0.000128152;
   DATA[2261,39] := 1.0;
   DATA[2261,40] := 1.0;
   DATA[2262,0] := 2.566698;
   DATA[2262,1] := 864.7775;
   DATA[2262,2] := 2.0;
   DATA[2262,3] := 2.0;
   DATA[2262,4] := 262.3366;
   DATA[2262,5] := 8.395475;
   DATA[2262,6] := 330.2999;
   DATA[2262,7] := 2.455003;
   DATA[2262,8] := 2.0;
   DATA[2262,9] := 2.0;
   DATA[2262,10] := 2.0;
   DATA[2262,11] := 19.70037;
   DATA[2262,12] := 2.209525;
   DATA[2262,13] := 811.9713;
   DATA[2262,14] := 1.0;
   DATA[2262,15] := 2.0;
   DATA[2262,16] := 1.0;
   DATA[2262,17] := 1.0;
   DATA[2262,18] := 1.0;
   DATA[2262,19] := 2.0;
   DATA[2262,20] := 148.808;
   DATA[2262,21] := 155.191;
   DATA[2262,22] := 1.719027;
   DATA[2262,23] := 848.8593;
   DATA[2262,24] := 2.0;
   DATA[2262,25] := 2.0;
   DATA[2262,26] := 7.874455;
   DATA[2262,27] := 144.3989;
   DATA[2262,28] := 261.7278;
   DATA[2262,29] := 11.95847;
   DATA[2262,30] := 1.728531;
   DATA[2262,31] := 1.266812;
   DATA[2262,32] := 0.7352687;
   DATA[2262,33] := 0.306761;
   DATA[2262,34] := 2.0;
   DATA[2262,35] := 250.3365;
   DATA[2262,36] := 1.681991;
   DATA[2262,37] := 189.1182;
   DATA[2262,38] := 0.000128152;
   DATA[2262,39] := 1.0;
   DATA[2262,40] := 1.0;
   DATA[2263,0] := 2.552285;
   DATA[2263,1] := 864.856;
   DATA[2263,2] := 2.0;
   DATA[2263,3] := 2.0;
   DATA[2263,4] := 262.3366;
   DATA[2263,5] := 8.395475;
   DATA[2263,6] := 330.2999;
   DATA[2263,7] := 2.455003;
   DATA[2263,8] := 2.0;
   DATA[2263,9] := 2.0;
   DATA[2263,10] := 2.0;
   DATA[2263,11] := 19.65555;
   DATA[2263,12] := 2.209013;
   DATA[2263,13] := 812.1315;
   DATA[2263,14] := 1.0;
   DATA[2263,15] := 2.0;
   DATA[2263,16] := 1.0;
   DATA[2263,17] := 1.0;
   DATA[2263,18] := 1.0;
   DATA[2263,19] := 2.0;
   DATA[2263,20] := 148.808;
   DATA[2263,21] := 155.191;
   DATA[2263,22] := 1.719027;
   DATA[2263,23] := 849.1669;
   DATA[2263,24] := 2.0;
   DATA[2263,25] := 2.0;
   DATA[2263,26] := 7.874455;
   DATA[2263,27] := 144.3476;
   DATA[2263,28] := 261.7278;
   DATA[2263,29] := 11.95847;
   DATA[2263,30] := 1.728531;
   DATA[2263,31] := 1.280902;
   DATA[2263,32] := 0.7352687;
   DATA[2263,33] := 0.306761;
   DATA[2263,34] := 2.0;
   DATA[2263,35] := 250.3365;
   DATA[2263,36] := 1.681991;
   DATA[2263,37] := 189.1182;
   DATA[2263,38] := 0.000128152;
   DATA[2263,39] := 1.0;
   DATA[2263,40] := 1.0;
   DATA[2264,0] := 2.536271;
   DATA[2264,1] := 864.9738;
   DATA[2264,2] := 2.0;
   DATA[2264,3] := 2.0;
   DATA[2264,4] := 262.3366;
   DATA[2264,5] := 8.395475;
   DATA[2264,6] := 330.2999;
   DATA[2264,7] := 2.456156;
   DATA[2264,8] := 2.0;
   DATA[2264,9] := 2.0;
   DATA[2264,10] := 2.0;
   DATA[2264,11] := 19.65555;
   DATA[2264,12] := 2.209013;
   DATA[2264,13] := 811.9713;
   DATA[2264,14] := 1.0;
   DATA[2264,15] := 2.0;
   DATA[2264,16] := 1.0;
   DATA[2264,17] := 1.0;
   DATA[2264,18] := 1.0;
   DATA[2264,19] := 2.0;
   DATA[2264,20] := 148.808;
   DATA[2264,21] := 155.191;
   DATA[2264,22] := 1.719027;
   DATA[2264,23] := 849.1669;
   DATA[2264,24] := 2.0;
   DATA[2264,25] := 2.0;
   DATA[2264,26] := 7.874455;
   DATA[2264,27] := 144.2194;
   DATA[2264,28] := 261.7278;
   DATA[2264,29] := 11.95847;
   DATA[2264,30] := 1.728531;
   DATA[2264,31] := 1.291277;
   DATA[2264,32] := 0.7352687;
   DATA[2264,33] := 0.3075937;
   DATA[2264,34] := 2.0;
   DATA[2264,35] := 250.3365;
   DATA[2264,36] := 1.681991;
   DATA[2264,37] := 189.1182;
   DATA[2264,38] := 0.000128152;
   DATA[2264,39] := 1.0;
   DATA[2264,40] := 1.0;
   DATA[2265,0] := 2.524101;
   DATA[2265,1] := 865.013;
   DATA[2265,2] := 2.0;
   DATA[2265,3] := 2.0;
   DATA[2265,4] := 262.3366;
   DATA[2265,5] := 8.395475;
   DATA[2265,6] := 330.223;
   DATA[2265,7] := 2.456541;
   DATA[2265,8] := 2.0;
   DATA[2265,9] := 2.0;
   DATA[2265,10] := 2.0;
   DATA[2265,11] := 19.65555;
   DATA[2265,12] := 2.209013;
   DATA[2265,13] := 811.8511;
   DATA[2265,14] := 1.0;
   DATA[2265,15] := 2.0;
   DATA[2265,16] := 1.0;
   DATA[2265,17] := 1.0;
   DATA[2265,18] := 1.0;
   DATA[2265,19] := 2.0;
   DATA[2265,20] := 148.808;
   DATA[2265,21] := 155.191;
   DATA[2265,22] := 1.717489;
   DATA[2265,23] := 849.7052;
   DATA[2265,24] := 2.0;
   DATA[2265,25] := 2.0;
   DATA[2265,26] := 7.874455;
   DATA[2265,27] := 144.2194;
   DATA[2265,28] := 261.7278;
   DATA[2265,29] := 11.95847;
   DATA[2265,30] := 1.728531;
   DATA[2265,31] := 1.308569;
   DATA[2265,32] := 0.7352687;
   DATA[2265,33] := 0.3082983;
   DATA[2265,34] := 2.0;
   DATA[2265,35] := 250.3365;
   DATA[2265,36] := 1.681991;
   DATA[2265,37] := 189.1182;
   DATA[2265,38] := 0.000128152;
   DATA[2265,39] := 1.0;
   DATA[2265,40] := 1.0;
   DATA[2266,0] := 2.504244;
   DATA[2266,1] := 864.6205;
   DATA[2266,2] := 2.0;
   DATA[2266,3] := 2.0;
   DATA[2266,4] := 262.3366;
   DATA[2266,5] := 8.395475;
   DATA[2266,6] := 330.1974;
   DATA[2266,7] := 2.457181;
   DATA[2266,8] := 2.0;
   DATA[2266,9] := 2.0;
   DATA[2266,10] := 2.0;
   DATA[2266,11] := 19.65555;
   DATA[2266,12] := 2.211959;
   DATA[2266,13] := 812.2116;
   DATA[2266,14] := 1.0;
   DATA[2266,15] := 2.0;
   DATA[2266,16] := 1.0;
   DATA[2266,17] := 1.0;
   DATA[2266,18] := 1.0;
   DATA[2266,19] := 2.0;
   DATA[2266,20] := 148.808;
   DATA[2266,21] := 155.0884;
   DATA[2266,22] := 1.717489;
   DATA[2266,23] := 849.5514;
   DATA[2266,24] := 2.0;
   DATA[2266,25] := 2.0;
   DATA[2266,26] := 7.874455;
   DATA[2266,27] := 144.2194;
   DATA[2266,28] := 261.7278;
   DATA[2266,29] := 11.95847;
   DATA[2266,30] := 1.728531;
   DATA[2266,31] := 1.30652;
   DATA[2266,32] := 0.7352687;
   DATA[2266,33] := 0.3082983;
   DATA[2266,34] := 2.0;
   DATA[2266,35] := 250.3365;
   DATA[2266,36] := 1.681991;
   DATA[2266,37] := 189.1182;
   DATA[2266,38] := 0.000128152;
   DATA[2266,39] := 1.0;
   DATA[2266,40] := 1.0;
   DATA[2267,0] := 2.485667;
   DATA[2267,1] := 864.7383;
   DATA[2267,2] := 2.0;
   DATA[2267,3] := 2.0;
   DATA[2267,4] := 262.3366;
   DATA[2267,5] := 8.395475;
   DATA[2267,6] := 330.1974;
   DATA[2267,7] := 2.457181;
   DATA[2267,8] := 2.0;
   DATA[2267,9] := 2.0;
   DATA[2267,10] := 2.0;
   DATA[2267,11] := 19.64594;
   DATA[2267,12] := 2.211959;
   DATA[2267,13] := 812.452;
   DATA[2267,14] := 1.0;
   DATA[2267,15] := 2.0;
   DATA[2267,16] := 1.0;
   DATA[2267,17] := 1.0;
   DATA[2267,18] := 1.0;
   DATA[2267,19] := 2.0;
   DATA[2267,20] := 148.808;
   DATA[2267,21] := 155.0884;
   DATA[2267,22] := 1.717489;
   DATA[2267,23] := 849.859;
   DATA[2267,24] := 2.0;
   DATA[2267,25] := 2.0;
   DATA[2267,26] := 7.874455;
   DATA[2267,27] := 144.2194;
   DATA[2267,28] := 261.7278;
   DATA[2267,29] := 11.95847;
   DATA[2267,30] := 1.729172;
   DATA[2267,31] := 1.3005;
   DATA[2267,32] := 0.7352687;
   DATA[2267,33] := 0.3082983;
   DATA[2267,34] := 2.0;
   DATA[2267,35] := 250.3365;
   DATA[2267,36] := 1.681991;
   DATA[2267,37] := 189.1182;
   DATA[2267,38] := 0.000128152;
   DATA[2267,39] := 1.0;
   DATA[2267,40] := 1.0;
   DATA[2268,0] := 2.471575;
   DATA[2268,1] := 864.385;
   DATA[2268,2] := 2.0;
   DATA[2268,3] := 2.0;
   DATA[2268,4] := 262.3366;
   DATA[2268,5] := 8.395475;
   DATA[2268,6] := 330.1974;
   DATA[2268,7] := 2.457181;
   DATA[2268,8] := 2.0;
   DATA[2268,9] := 2.0;
   DATA[2268,10] := 2.0;
   DATA[2268,11] := 19.62354;
   DATA[2268,12] := 2.211959;
   DATA[2268,13] := 812.6522;
   DATA[2268,14] := 1.0;
   DATA[2268,15] := 2.0;
   DATA[2268,16] := 1.0;
   DATA[2268,17] := 1.0;
   DATA[2268,18] := 1.0;
   DATA[2268,19] := 2.0;
   DATA[2268,20] := 148.808;
   DATA[2268,21] := 155.0884;
   DATA[2268,22] := 1.717489;
   DATA[2268,23] := 849.8975;
   DATA[2268,24] := 2.0;
   DATA[2268,25] := 2.0;
   DATA[2268,26] := 7.874455;
   DATA[2268,27] := 144.2194;
   DATA[2268,28] := 261.7278;
   DATA[2268,29] := 11.95847;
   DATA[2268,30] := 1.729172;
   DATA[2268,31] := 1.293839;
   DATA[2268,32] := 0.7352687;
   DATA[2268,33] := 0.3086827;
   DATA[2268,34] := 2.0;
   DATA[2268,35] := 250.3365;
   DATA[2268,36] := 1.681991;
   DATA[2268,37] := 189.1182;
   DATA[2268,38] := 0.000128152;
   DATA[2268,39] := 1.0;
   DATA[2268,40] := 1.0;
   DATA[2269,0] := 2.45364;
   DATA[2269,1] := 864.6205;
   DATA[2269,2] := 2.0;
   DATA[2269,3] := 2.0;
   DATA[2269,4] := 262.3366;
   DATA[2269,5] := 8.395475;
   DATA[2269,6] := 330.1974;
   DATA[2269,7] := 2.457181;
   DATA[2269,8] := 2.0;
   DATA[2269,9] := 2.0;
   DATA[2269,10] := 2.0;
   DATA[2269,11] := 19.62354;
   DATA[2269,12] := 2.210806;
   DATA[2269,13] := 812.7724;
   DATA[2269,14] := 1.0;
   DATA[2269,15] := 2.0;
   DATA[2269,16] := 1.0;
   DATA[2269,17] := 1.0;
   DATA[2269,18] := 1.0;
   DATA[2269,19] := 2.0;
   DATA[2269,20] := 148.808;
   DATA[2269,21] := 155.0884;
   DATA[2269,22] := 1.718771;
   DATA[2269,23] := 850.0897;
   DATA[2269,24] := 2.0;
   DATA[2269,25] := 2.0;
   DATA[2269,26] := 7.874455;
   DATA[2269,27] := 144.2194;
   DATA[2269,28] := 261.7278;
   DATA[2269,29] := 11.95847;
   DATA[2269,30] := 1.729172;
   DATA[2269,31] := 1.282823;
   DATA[2269,32] := 0.7352687;
   DATA[2269,33] := 0.3086827;
   DATA[2269,34] := 2.0;
   DATA[2269,35] := 250.4166;
   DATA[2269,36] := 1.681991;
   DATA[2269,37] := 189.2784;
   DATA[2269,38] := 0.000128152;
   DATA[2269,39] := 1.0;
   DATA[2269,40] := 1.0;
   DATA[2270,0] := 2.436985;
   DATA[2270,1] := 864.4635;
   DATA[2270,2] := 2.0;
   DATA[2270,3] := 2.0;
   DATA[2270,4] := 262.3366;
   DATA[2270,5] := 8.395475;
   DATA[2270,6] := 330.1974;
   DATA[2270,7] := 2.457181;
   DATA[2270,8] := 2.0;
   DATA[2270,9] := 2.0;
   DATA[2270,10] := 2.0;
   DATA[2270,11] := 19.68436;
   DATA[2270,12] := 2.208884;
   DATA[2270,13] := 812.9326;
   DATA[2270,14] := 1.0;
   DATA[2270,15] := 2.0;
   DATA[2270,16] := 1.0;
   DATA[2270,17] := 1.0;
   DATA[2270,18] := 1.0;
   DATA[2270,19] := 2.0;
   DATA[2270,20] := 148.808;
   DATA[2270,21] := 155.0884;
   DATA[2270,22] := 1.718771;
   DATA[2270,23] := 850.0897;
   DATA[2270,24] := 2.0;
   DATA[2270,25] := 2.0;
   DATA[2270,26] := 7.874455;
   DATA[2270,27] := 144.2194;
   DATA[2270,28] := 261.7278;
   DATA[2270,29] := 11.95847;
   DATA[2270,30] := 1.729172;
   DATA[2270,31] := 1.282567;
   DATA[2270,32] := 0.7352687;
   DATA[2270,33] := 0.3086827;
   DATA[2270,34] := 2.0;
   DATA[2270,35] := 250.5127;
   DATA[2270,36] := 1.681991;
   DATA[2270,37] := 189.2944;
   DATA[2270,38] := 0.000128152;
   DATA[2270,39] := 1.0;
   DATA[2270,40] := 1.0;
   DATA[2271,0] := 2.425135;
   DATA[2271,1] := 864.385;
   DATA[2271,2] := 2.0;
   DATA[2271,3] := 2.0;
   DATA[2271,4] := 262.3366;
   DATA[2271,5] := 8.395475;
   DATA[2271,6] := 330.1974;
   DATA[2271,7] := 2.457181;
   DATA[2271,8] := 2.0;
   DATA[2271,9] := 2.0;
   DATA[2271,10] := 2.0;
   DATA[2271,11] := 19.70037;
   DATA[2271,12] := 2.208884;
   DATA[2271,13] := 812.9326;
   DATA[2271,14] := 1.0;
   DATA[2271,15] := 2.0;
   DATA[2271,16] := 1.0;
   DATA[2271,17] := 1.0;
   DATA[2271,18] := 1.0;
   DATA[2271,19] := 2.0;
   DATA[2271,20] := 148.808;
   DATA[2271,21] := 155.0884;
   DATA[2271,22] := 1.718771;
   DATA[2271,23] := 850.2051;
   DATA[2271,24] := 2.0;
   DATA[2271,25] := 2.0;
   DATA[2271,26] := 7.874455;
   DATA[2271,27] := 144.2194;
   DATA[2271,28] := 261.7278;
   DATA[2271,29] := 11.95847;
   DATA[2271,30] := 1.729172;
   DATA[2271,31] := 1.292046;
   DATA[2271,32] := 0.7352687;
   DATA[2271,33] := 0.3074016;
   DATA[2271,34] := 2.0;
   DATA[2271,35] := 250.5127;
   DATA[2271,36] := 1.681991;
   DATA[2271,37] := 189.3265;
   DATA[2271,38] := 0.000128152;
   DATA[2271,39] := 1.0;
   DATA[2271,40] := 1.0;
   DATA[2272,0] := 2.422573;
   DATA[2272,1] := 864.2672;
   DATA[2272,2] := 2.0;
   DATA[2272,3] := 2.0;
   DATA[2272,4] := 262.3366;
   DATA[2272,5] := 8.395475;
   DATA[2272,6] := 330.1974;
   DATA[2272,7] := 2.457181;
   DATA[2272,8] := 2.0;
   DATA[2272,9] := 2.0;
   DATA[2272,10] := 2.0;
   DATA[2272,11] := 19.70037;
   DATA[2272,12] := 2.208884;
   DATA[2272,13] := 812.9727;
   DATA[2272,14] := 1.0;
   DATA[2272,15] := 2.0;
   DATA[2272,16] := 1.0;
   DATA[2272,17] := 1.0;
   DATA[2272,18] := 1.0;
   DATA[2272,19] := 2.0;
   DATA[2272,20] := 148.808;
   DATA[2272,21] := 155.0884;
   DATA[2272,22] := 1.718771;
   DATA[2272,23] := 850.282;
   DATA[2272,24] := 2.0;
   DATA[2272,25] := 2.0;
   DATA[2272,26] := 7.874455;
   DATA[2272,27] := 144.2194;
   DATA[2272,28] := 261.7278;
   DATA[2272,29] := 11.95847;
   DATA[2272,30] := 1.728916;
   DATA[2272,31] := 1.292046;
   DATA[2272,32] := 0.7355248;
   DATA[2272,33] := 0.3070813;
   DATA[2272,34] := 2.0;
   DATA[2272,35] := 250.5127;
   DATA[2272,36] := 1.681991;
   DATA[2272,37] := 189.3265;
   DATA[2272,38] := 0.000128152;
   DATA[2272,39] := 1.0;
   DATA[2272,40] := 1.0;
   DATA[2273,0] := 2.422573;
   DATA[2273,1] := 864.1495;
   DATA[2273,2] := 2.0;
   DATA[2273,3] := 2.0;
   DATA[2273,4] := 262.3366;
   DATA[2273,5] := 8.395475;
   DATA[2273,6] := 330.1974;
   DATA[2273,7] := 2.457181;
   DATA[2273,8] := 2.0;
   DATA[2273,9] := 2.0;
   DATA[2273,10] := 2.0;
   DATA[2273,11] := 19.70037;
   DATA[2273,12] := 2.20645;
   DATA[2273,13] := 813.1329;
   DATA[2273,14] := 1.0;
   DATA[2273,15] := 2.0;
   DATA[2273,16] := 1.0;
   DATA[2273,17] := 1.0;
   DATA[2273,18] := 1.0;
   DATA[2273,19] := 2.0;
   DATA[2273,20] := 148.808;
   DATA[2273,21] := 155.0884;
   DATA[2273,22] := 1.718771;
   DATA[2273,23] := 850.5127;
   DATA[2273,24] := 2.0;
   DATA[2273,25] := 2.0;
   DATA[2273,26] := 7.874455;
   DATA[2273,27] := 144.2194;
   DATA[2273,28] := 261.7278;
   DATA[2273,29] := 11.95847;
   DATA[2273,30] := 1.728659;
   DATA[2273,31] := 1.298962;
   DATA[2273,32] := 0.7355248;
   DATA[2273,33] := 0.3068891;
   DATA[2273,34] := 2.0;
   DATA[2273,35] := 250.5127;
   DATA[2273,36] := 1.681991;
   DATA[2273,37] := 189.3265;
   DATA[2273,38] := 0.000128152;
   DATA[2273,39] := 1.0;
   DATA[2273,40] := 1.0;
   DATA[2274,0] := 2.439868;
   DATA[2274,1] := 864.6205;
   DATA[2274,2] := 2.0;
   DATA[2274,3] := 2.0;
   DATA[2274,4] := 262.3366;
   DATA[2274,5] := 8.395475;
   DATA[2274,6] := 330.0436;
   DATA[2274,7] := 2.457181;
   DATA[2274,8] := 2.0;
   DATA[2274,9] := 2.0;
   DATA[2274,10] := 2.0;
   DATA[2274,11] := 19.70037;
   DATA[2274,12] := 2.20645;
   DATA[2274,13] := 813.213;
   DATA[2274,14] := 1.0;
   DATA[2274,15] := 2.0;
   DATA[2274,16] := 1.0;
   DATA[2274,17] := 1.0;
   DATA[2274,18] := 1.0;
   DATA[2274,19] := 2.0;
   DATA[2274,20] := 148.808;
   DATA[2274,21] := 155.0884;
   DATA[2274,22] := 1.719284;
   DATA[2274,23] := 850.6281;
   DATA[2274,24] := 2.0;
   DATA[2274,25] := 2.0;
   DATA[2274,26] := 7.874455;
   DATA[2274,27] := 144.2194;
   DATA[2274,28] := 261.7278;
   DATA[2274,29] := 11.95847;
   DATA[2274,30] := 1.727634;
   DATA[2274,31] := 1.306008;
   DATA[2274,32] := 0.7355248;
   DATA[2274,33] := 0.3065048;
   DATA[2274,34] := 2.0;
   DATA[2274,35] := 250.5127;
   DATA[2274,36] := 1.681991;
   DATA[2274,37] := 189.3265;
   DATA[2274,38] := 0.000128152;
   DATA[2274,39] := 1.0;
   DATA[2274,40] := 1.0;
   DATA[2275,0] := 2.484066;
   DATA[2275,1] := 864.3457;
   DATA[2275,2] := 2.0;
   DATA[2275,3] := 2.0;
   DATA[2275,4] := 262.3366;
   DATA[2275,5] := 8.395475;
   DATA[2275,6] := 330.0436;
   DATA[2275,7] := 2.457181;
   DATA[2275,8] := 2.0;
   DATA[2275,9] := 2.0;
   DATA[2275,10] := 2.0;
   DATA[2275,11] := 19.70037;
   DATA[2275,12] := 2.207988;
   DATA[2275,13] := 813.1729;
   DATA[2275,14] := 1.0;
   DATA[2275,15] := 2.0;
   DATA[2275,16] := 1.0;
   DATA[2275,17] := 1.0;
   DATA[2275,18] := 1.0;
   DATA[2275,19] := 2.0;
   DATA[2275,20] := 148.808;
   DATA[2275,21] := 155.0884;
   DATA[2275,22] := 1.719284;
   DATA[2275,23] := 850.3204;
   DATA[2275,24] := 2.0;
   DATA[2275,25] := 2.0;
   DATA[2275,26] := 7.874455;
   DATA[2275,27] := 144.2194;
   DATA[2275,28] := 261.7278;
   DATA[2275,29] := 11.95847;
   DATA[2275,30] := 1.727634;
   DATA[2275,31] := 1.287562;
   DATA[2275,32] := 0.7355248;
   DATA[2275,33] := 0.3065048;
   DATA[2275,34] := 2.0;
   DATA[2275,35] := 250.5127;
   DATA[2275,36] := 1.681991;
   DATA[2275,37] := 189.3265;
   DATA[2275,38] := 0.000128152;
   DATA[2275,39] := 1.0;
   DATA[2275,40] := 1.0;
   DATA[2276,0] := 2.525702;
   DATA[2276,1] := 864.071;
   DATA[2276,2] := 2.0;
   DATA[2276,3] := 2.0;
   DATA[2276,4] := 262.3366;
   DATA[2276,5] := 8.395475;
   DATA[2276,6] := 330.0436;
   DATA[2276,7] := 2.457181;
   DATA[2276,8] := 2.0;
   DATA[2276,9] := 2.0;
   DATA[2276,10] := 2.0;
   DATA[2276,11] := 19.73558;
   DATA[2276,12] := 2.209013;
   DATA[2276,13] := 813.213;
   DATA[2276,14] := 1.0;
   DATA[2276,15] := 2.0;
   DATA[2276,16] := 1.0;
   DATA[2276,17] := 1.0;
   DATA[2276,18] := 1.0;
   DATA[2276,19] := 2.0;
   DATA[2276,20] := 148.808;
   DATA[2276,21] := 155.0884;
   DATA[2276,22] := 1.719284;
   DATA[2276,23] := 850.282;
   DATA[2276,24] := 2.0;
   DATA[2276,25] := 2.0;
   DATA[2276,26] := 7.874455;
   DATA[2276,27] := 144.322;
   DATA[2276,28] := 261.7278;
   DATA[2276,29] := 11.95847;
   DATA[2276,30] := 1.727634;
   DATA[2276,31] := 1.281798;
   DATA[2276,32] := 0.7355248;
   DATA[2276,33] := 0.3065048;
   DATA[2276,34] := 2.0;
   DATA[2276,35] := 250.5127;
   DATA[2276,36] := 1.681991;
   DATA[2276,37] := 189.3265;
   DATA[2276,38] := 0.000128152;
   DATA[2276,39] := 1.0;
   DATA[2276,40] := 1.0;
   DATA[2277,0] := 2.571182;
   DATA[2277,1] := 863.9924;
   DATA[2277,2] := 2.0;
   DATA[2277,3] := 2.0;
   DATA[2277,4] := 262.3366;
   DATA[2277,5] := 8.395475;
   DATA[2277,6] := 330.0436;
   DATA[2277,7] := 2.455643;
   DATA[2277,8] := 2.0;
   DATA[2277,9] := 2.0;
   DATA[2277,10] := 2.0;
   DATA[2277,11] := 19.73558;
   DATA[2277,12] := 2.209013;
   DATA[2277,13] := 813.0527;
   DATA[2277,14] := 1.0;
   DATA[2277,15] := 2.0;
   DATA[2277,16] := 1.0;
   DATA[2277,17] := 1.0;
   DATA[2277,18] := 1.0;
   DATA[2277,19] := 2.0;
   DATA[2277,20] := 148.808;
   DATA[2277,21] := 155.0884;
   DATA[2277,22] := 1.719156;
   DATA[2277,23] := 850.5127;
   DATA[2277,24] := 2.0;
   DATA[2277,25] := 2.0;
   DATA[2277,26] := 7.874455;
   DATA[2277,27] := 144.322;
   DATA[2277,28] := 261.7278;
   DATA[2277,29] := 11.95847;
   DATA[2277,30] := 1.728531;
   DATA[2277,31] := 1.266299;
   DATA[2277,32] := 0.7355248;
   DATA[2277,33] := 0.3065048;
   DATA[2277,34] := 2.0;
   DATA[2277,35] := 250.5127;
   DATA[2277,36] := 1.681991;
   DATA[2277,37] := 189.3265;
   DATA[2277,38] := 0.000128152;
   DATA[2277,39] := 1.0;
   DATA[2277,40] := 1.0;
   DATA[2278,0] := 2.611216;
   DATA[2278,1] := 863.757;
   DATA[2278,2] := 2.0;
   DATA[2278,3] := 2.0;
   DATA[2278,4] := 262.3366;
   DATA[2278,5] := 8.395475;
   DATA[2278,6] := 330.0436;
   DATA[2278,7] := 2.455643;
   DATA[2278,8] := 2.0;
   DATA[2278,9] := 2.0;
   DATA[2278,10] := 2.0;
   DATA[2278,11] := 19.73558;
   DATA[2278,12] := 2.209013;
   DATA[2278,13] := 813.3331;
   DATA[2278,14] := 1.0;
   DATA[2278,15] := 2.0;
   DATA[2278,16] := 1.0;
   DATA[2278,17] := 1.0;
   DATA[2278,18] := 1.0;
   DATA[2278,19] := 2.0;
   DATA[2278,20] := 148.808;
   DATA[2278,21] := 155.0884;
   DATA[2278,22] := 1.717361;
   DATA[2278,23] := 850.8588;
   DATA[2278,24] := 2.0;
   DATA[2278,25] := 2.0;
   DATA[2278,26] := 7.874455;
   DATA[2278,27] := 144.322;
   DATA[2278,28] := 261.7278;
   DATA[2278,29] := 12.07383;
   DATA[2278,30] := 1.728659;
   DATA[2278,31] := 1.266428;
   DATA[2278,32] := 0.7355248;
   DATA[2278,33] := 0.3065048;
   DATA[2278,34] := 2.0;
   DATA[2278,35] := 250.4166;
   DATA[2278,36] := 1.681991;
   DATA[2278,37] := 189.3265;
   DATA[2278,38] := 0.000128152;
   DATA[2278,39] := 1.0;
   DATA[2278,40] := 1.0;
   DATA[2279,0] := 2.644205;
   DATA[2279,1] := 864.1887;
   DATA[2279,2] := 2.0;
   DATA[2279,3] := 2.0;
   DATA[2279,4] := 262.3366;
   DATA[2279,5] := 8.395475;
   DATA[2279,6] := 330.0436;
   DATA[2279,7] := 2.457181;
   DATA[2279,8] := 2.0;
   DATA[2279,9] := 2.0;
   DATA[2279,10] := 2.0;
   DATA[2279,11] := 19.68756;
   DATA[2279,12] := 2.209013;
   DATA[2279,13] := 812.8124;
   DATA[2279,14] := 1.0;
   DATA[2279,15] := 2.0;
   DATA[2279,16] := 1.0;
   DATA[2279,17] := 1.0;
   DATA[2279,18] := 1.0;
   DATA[2279,19] := 2.0;
   DATA[2279,20] := 148.808;
   DATA[2279,21] := 155.0884;
   DATA[2279,22] := 1.717361;
   DATA[2279,23] := 850.6665;
   DATA[2279,24] := 2.0;
   DATA[2279,25] := 2.0;
   DATA[2279,26] := 7.874455;
   DATA[2279,27] := 144.322;
   DATA[2279,28] := 261.7278;
   DATA[2279,29] := 12.30454;
   DATA[2279,30] := 1.728659;
   DATA[2279,31] := 1.280646;
   DATA[2279,32] := 0.7355248;
   DATA[2279,33] := 0.3065048;
   DATA[2279,34] := 2.0;
   DATA[2279,35] := 250.2724;
   DATA[2279,36] := 1.681991;
   DATA[2279,37] := 189.2944;
   DATA[2279,38] := 0.000128152;
   DATA[2279,39] := 1.0;
   DATA[2279,40] := 1.0;
   DATA[2280,0] := 2.657336;
   DATA[2280,1] := 864.1887;
   DATA[2280,2] := 2.0;
   DATA[2280,3] := 2.0;
   DATA[2280,4] := 262.3366;
   DATA[2280,5] := 8.395475;
   DATA[2280,6] := 330.0436;
   DATA[2280,7] := 2.457694;
   DATA[2280,8] := 2.0;
   DATA[2280,9] := 2.0;
   DATA[2280,10] := 2.0;
   DATA[2280,11] := 19.68756;
   DATA[2280,12] := 2.209013;
   DATA[2280,13] := 812.9727;
   DATA[2280,14] := 1.0;
   DATA[2280,15] := 2.0;
   DATA[2280,16] := 1.0;
   DATA[2280,17] := 1.0;
   DATA[2280,18] := 1.0;
   DATA[2280,19] := 2.0;
   DATA[2280,20] := 148.808;
   DATA[2280,21] := 155.0884;
   DATA[2280,22] := 1.717361;
   DATA[2280,23] := 850.8588;
   DATA[2280,24] := 2.0;
   DATA[2280,25] := 2.0;
   DATA[2280,26] := 7.874455;
   DATA[2280,27] := 144.322;
   DATA[2280,28] := 261.7278;
   DATA[2280,29] := 12.30454;
   DATA[2280,30] := 1.726993;
   DATA[2280,31] := 1.291277;
   DATA[2280,32] := 0.7355248;
   DATA[2280,33] := 0.3065048;
   DATA[2280,34] := 2.0;
   DATA[2280,35] := 250.2724;
   DATA[2280,36] := 1.681991;
   DATA[2280,37] := 189.1662;
   DATA[2280,38] := 0.000128152;
   DATA[2280,39] := 1.0;
   DATA[2280,40] := 1.0;
   DATA[2281,0] := 2.66182;
   DATA[2281,1] := 864.4635;
   DATA[2281,2] := 2.0;
   DATA[2281,3] := 2.0;
   DATA[2281,4] := 262.3366;
   DATA[2281,5] := 8.395475;
   DATA[2281,6] := 330.0436;
   DATA[2281,7] := 2.457694;
   DATA[2281,8] := 2.0;
   DATA[2281,9] := 2.0;
   DATA[2281,10] := 2.0;
   DATA[2281,11] := 19.76439;
   DATA[2281,12] := 2.209013;
   DATA[2281,13] := 812.8525;
   DATA[2281,14] := 1.0;
   DATA[2281,15] := 2.0;
   DATA[2281,16] := 1.0;
   DATA[2281,17] := 1.0;
   DATA[2281,18] := 1.0;
   DATA[2281,19] := 2.0;
   DATA[2281,20] := 148.808;
   DATA[2281,21] := 155.0884;
   DATA[2281,22] := 1.717361;
   DATA[2281,23] := 850.8972;
   DATA[2281,24] := 2.0;
   DATA[2281,25] := 2.0;
   DATA[2281,26] := 7.874455;
   DATA[2281,27] := 144.322;
   DATA[2281,28] := 261.7278;
   DATA[2281,29] := 12.30454;
   DATA[2281,30] := 1.726737;
   DATA[2281,31] := 1.302165;
   DATA[2281,32] := 0.7355248;
   DATA[2281,33] := 0.3083624;
   DATA[2281,34] := 2.0;
   DATA[2281,35] := 250.2724;
   DATA[2281,36] := 1.681991;
   DATA[2281,37] := 189.1662;
   DATA[2281,38] := 0.000128152;
   DATA[2281,39] := 1.0;
   DATA[2281,40] := 1.0;
   DATA[2282,0] := 2.646126;
   DATA[2282,1] := 864.6205;
   DATA[2282,2] := 2.0;
   DATA[2282,3] := 2.0;
   DATA[2282,4] := 262.3366;
   DATA[2282,5] := 8.395475;
   DATA[2282,6] := 330.0948;
   DATA[2282,7] := 2.457181;
   DATA[2282,8] := 2.0;
   DATA[2282,9] := 2.0;
   DATA[2282,10] := 2.0;
   DATA[2282,11] := 19.76439;
   DATA[2282,12] := 2.209525;
   DATA[2282,13] := 812.7724;
   DATA[2282,14] := 1.0;
   DATA[2282,15] := 2.0;
   DATA[2282,16] := 1.0;
   DATA[2282,17] := 1.0;
   DATA[2282,18] := 1.0;
   DATA[2282,19] := 2.0;
   DATA[2282,20] := 148.808;
   DATA[2282,21] := 155.0884;
   DATA[2282,22] := 1.717361;
   DATA[2282,23] := 850.8972;
   DATA[2282,24] := 2.0;
   DATA[2282,25] := 2.0;
   DATA[2282,26] := 7.874455;
   DATA[2282,27] := 144.322;
   DATA[2282,28] := 261.7278;
   DATA[2282,29] := 12.15073;
   DATA[2282,30] := 1.726737;
   DATA[2282,31] := 1.296657;
   DATA[2282,32] := 0.7355248;
   DATA[2282,33] := 0.3083624;
   DATA[2282,34] := 2.0;
   DATA[2282,35] := 250.2724;
   DATA[2282,36] := 1.681991;
   DATA[2282,37] := 189.1662;
   DATA[2282,38] := 0.000128152;
   DATA[2282,39] := 1.0;
   DATA[2282,40] := 1.0;
   DATA[2283,0] := 2.632995;
   DATA[2283,1] := 864.542;
   DATA[2283,2] := 2.0;
   DATA[2283,3] := 2.0;
   DATA[2283,4] := 262.3366;
   DATA[2283,5] := 8.395475;
   DATA[2283,6] := 330.0948;
   DATA[2283,7] := 2.457181;
   DATA[2283,8] := 2.0;
   DATA[2283,9] := 2.0;
   DATA[2283,10] := 2.0;
   DATA[2283,11] := 19.76439;
   DATA[2283,12] := 2.21055;
   DATA[2283,13] := 812.9727;
   DATA[2283,14] := 1.0;
   DATA[2283,15] := 2.0;
   DATA[2283,16] := 1.0;
   DATA[2283,17] := 1.0;
   DATA[2283,18] := 1.0;
   DATA[2283,19] := 2.0;
   DATA[2283,20] := 148.808;
   DATA[2283,21] := 155.0884;
   DATA[2283,22] := 1.717361;
   DATA[2283,23] := 850.8588;
   DATA[2283,24] := 2.0;
   DATA[2283,25] := 2.0;
   DATA[2283,26] := 7.874455;
   DATA[2283,27] := 144.322;
   DATA[2283,28] := 261.7278;
   DATA[2283,29] := 12.15073;
   DATA[2283,30] := 1.726993;
   DATA[2283,31] := 1.282311;
   DATA[2283,32] := 0.7355248;
   DATA[2283,33] := 0.3083624;
   DATA[2283,34] := 2.0;
   DATA[2283,35] := 250.2724;
   DATA[2283,36] := 1.681991;
   DATA[2283,37] := 189.1662;
   DATA[2283,38] := 0.000128152;
   DATA[2283,39] := 1.0;
   DATA[2283,40] := 1.0;
   DATA[2284,0] := 2.625628;
   DATA[2284,1] := 864.856;
   DATA[2284,2] := 2.0;
   DATA[2284,3] := 2.0;
   DATA[2284,4] := 262.3366;
   DATA[2284,5] := 8.395475;
   DATA[2284,6] := 330.0948;
   DATA[2284,7] := 2.457181;
   DATA[2284,8] := 2.0;
   DATA[2284,9] := 2.0;
   DATA[2284,10] := 2.0;
   DATA[2284,11] := 19.76439;
   DATA[2284,12] := 2.21055;
   DATA[2284,13] := 812.7324;
   DATA[2284,14] := 1.0;
   DATA[2284,15] := 2.0;
   DATA[2284,16] := 1.0;
   DATA[2284,17] := 1.0;
   DATA[2284,18] := 1.0;
   DATA[2284,19] := 2.0;
   DATA[2284,20] := 148.808;
   DATA[2284,21] := 155.0884;
   DATA[2284,22] := 1.718771;
   DATA[2284,23] := 851.0126;
   DATA[2284,24] := 2.0;
   DATA[2284,25] := 2.0;
   DATA[2284,26] := 7.874455;
   DATA[2284,27] := 144.322;
   DATA[2284,28] := 261.7278;
   DATA[2284,29] := 11.95847;
   DATA[2284,30] := 1.726993;
   DATA[2284,31] := 1.282183;
   DATA[2284,32] := 0.7355248;
   DATA[2284,33] := 0.3083624;
   DATA[2284,34] := 2.0;
   DATA[2284,35] := 250.2724;
   DATA[2284,36] := 1.681991;
   DATA[2284,37] := 189.1662;
   DATA[2284,38] := 0.000128152;
   DATA[2284,39] := 1.0;
   DATA[2284,40] := 1.0;
   DATA[2285,0] := 2.618903;
   DATA[2285,1] := 865.013;
   DATA[2285,2] := 2.0;
   DATA[2285,3] := 2.0;
   DATA[2285,4] := 262.3366;
   DATA[2285,5] := 8.395475;
   DATA[2285,6] := 330.0948;
   DATA[2285,7] := 2.457053;
   DATA[2285,8] := 2.0;
   DATA[2285,9] := 2.0;
   DATA[2285,10] := 2.0;
   DATA[2285,11] := 19.74198;
   DATA[2285,12] := 2.21055;
   DATA[2285,13] := 813.1329;
   DATA[2285,14] := 1.0;
   DATA[2285,15] := 2.0;
   DATA[2285,16] := 1.0;
   DATA[2285,17] := 1.0;
   DATA[2285,18] := 1.0;
   DATA[2285,19] := 2.0;
   DATA[2285,20] := 148.808;
   DATA[2285,21] := 155.0628;
   DATA[2285,22] := 1.719027;
   DATA[2285,23] := 850.5896;
   DATA[2285,24] := 2.0;
   DATA[2285,25] := 2.0;
   DATA[2285,26] := 7.874455;
   DATA[2285,27] := 144.527;
   DATA[2285,28] := 261.7278;
   DATA[2285,29] := 11.95847;
   DATA[2285,30] := 1.729172;
   DATA[2285,31] := 1.271935;
   DATA[2285,32] := 0.7355248;
   DATA[2285,33] := 0.3083624;
   DATA[2285,34] := 2.0;
   DATA[2285,35] := 250.4005;
   DATA[2285,36] := 1.681991;
   DATA[2285,37] := 189.1662;
   DATA[2285,38] := 0.000128152;
   DATA[2285,39] := 1.0;
   DATA[2285,40] := 1.0;
   DATA[2286,0] := 2.607693;
   DATA[2286,1] := 864.9345;
   DATA[2286,2] := 2.0;
   DATA[2286,3] := 2.0;
   DATA[2286,4] := 262.3366;
   DATA[2286,5] := 8.395475;
   DATA[2286,6] := 330.0948;
   DATA[2286,7] := 2.4559;
   DATA[2286,8] := 2.0;
   DATA[2286,9] := 2.0;
   DATA[2286,10] := 2.0;
   DATA[2286,11] := 19.74198;
   DATA[2286,12] := 2.21055;
   DATA[2286,13] := 812.9326;
   DATA[2286,14] := 1.0;
   DATA[2286,15] := 2.0;
   DATA[2286,16] := 1.0;
   DATA[2286,17] := 1.0;
   DATA[2286,18] := 1.0;
   DATA[2286,19] := 2.0;
   DATA[2286,20] := 148.808;
   DATA[2286,21] := 154.9603;
   DATA[2286,22] := 1.720693;
   DATA[2286,23] := 850.8588;
   DATA[2286,24] := 2.0;
   DATA[2286,25] := 2.0;
   DATA[2286,26] := 7.874455;
   DATA[2286,27] := 144.527;
   DATA[2286,28] := 261.7278;
   DATA[2286,29] := 11.95847;
   DATA[2286,30] := 1.729428;
   DATA[2286,31] := 1.262329;
   DATA[2286,32] := 0.7355248;
   DATA[2286,33] := 0.3083624;
   DATA[2286,34] := 2.0;
   DATA[2286,35] := 250.4005;
   DATA[2286,36] := 1.681991;
   DATA[2286,37] := 189.2944;
   DATA[2286,38] := 0.000128152;
   DATA[2286,39] := 1.0;
   DATA[2286,40] := 1.0;
   DATA[2287,0] := 2.582391;
   DATA[2287,1] := 864.7775;
   DATA[2287,2] := 2.0;
   DATA[2287,3] := 2.0;
   DATA[2287,4] := 262.3366;
   DATA[2287,5] := 8.395475;
   DATA[2287,6] := 330.0948;
   DATA[2287,7] := 2.453337;
   DATA[2287,8] := 2.0;
   DATA[2287,9] := 2.0;
   DATA[2287,10] := 2.0;
   DATA[2287,11] := 19.73238;
   DATA[2287,12] := 2.21055;
   DATA[2287,13] := 813.3732;
   DATA[2287,14] := 1.0;
   DATA[2287,15] := 2.0;
   DATA[2287,16] := 1.0;
   DATA[2287,17] := 1.0;
   DATA[2287,18] := 1.0;
   DATA[2287,19] := 2.0;
   DATA[2287,20] := 148.808;
   DATA[2287,21] := 154.909;
   DATA[2287,22] := 1.720693;
   DATA[2287,23] := 850.6665;
   DATA[2287,24] := 2.0;
   DATA[2287,25] := 2.0;
   DATA[2287,26] := 7.874455;
   DATA[2287,27] := 144.527;
   DATA[2287,28] := 261.7278;
   DATA[2287,29] := 11.95847;
   DATA[2287,30] := 1.729428;
   DATA[2287,31] := 1.271679;
   DATA[2287,32] := 0.7355248;
   DATA[2287,33] := 0.3083624;
   DATA[2287,34] := 2.0;
   DATA[2287,35] := 250.4005;
   DATA[2287,36] := 1.681991;
   DATA[2287,37] := 189.2944;
   DATA[2287,38] := 0.000128152;
   DATA[2287,39] := 1.0;
   DATA[2287,40] := 1.0;
   DATA[2288,0] := 2.564776;
   DATA[2288,1] := 864.542;
   DATA[2288,2] := 2.0;
   DATA[2288,3] := 2.0;
   DATA[2288,4] := 262.3366;
   DATA[2288,5] := 8.395475;
   DATA[2288,6] := 330.0948;
   DATA[2288,7] := 2.45308;
   DATA[2288,8] := 2.0;
   DATA[2288,9] := 2.0;
   DATA[2288,10] := 2.0;
   DATA[2288,11] := 19.73238;
   DATA[2288,12] := 2.210037;
   DATA[2288,13] := 813.0527;
   DATA[2288,14] := 1.0;
   DATA[2288,15] := 2.0;
   DATA[2288,16] := 1.0;
   DATA[2288,17] := 1.0;
   DATA[2288,18] := 1.0;
   DATA[2288,19] := 2.0;
   DATA[2288,20] := 148.808;
   DATA[2288,21] := 154.909;
   DATA[2288,22] := 1.720693;
   DATA[2288,23] := 850.8203;
   DATA[2288,24] := 2.0;
   DATA[2288,25] := 2.0;
   DATA[2288,26] := 7.874455;
   DATA[2288,27] := 144.527;
   DATA[2288,28] := 261.7278;
   DATA[2288,29] := 11.95847;
   DATA[2288,30] := 1.730838;
   DATA[2288,31] := 1.289356;
   DATA[2288,32] := 0.7355248;
   DATA[2288,33] := 0.3083624;
   DATA[2288,34] := 2.0;
   DATA[2288,35] := 250.4005;
   DATA[2288,36] := 1.681991;
   DATA[2288,37] := 189.2944;
   DATA[2288,38] := 0.000128152;
   DATA[2288,39] := 1.0;
   DATA[2288,40] := 1.0;
   DATA[2289,0] := 2.548121;
   DATA[2289,1] := 864.7383;
   DATA[2289,2] := 2.0;
   DATA[2289,3] := 2.0;
   DATA[2289,4] := 262.3366;
   DATA[2289,5] := 8.395475;
   DATA[2289,6] := 330.0948;
   DATA[2289,7] := 2.454875;
   DATA[2289,8] := 2.0;
   DATA[2289,9] := 2.0;
   DATA[2289,10] := 2.0;
   DATA[2289,11] := 19.73238;
   DATA[2289,12] := 2.209269;
   DATA[2289,13] := 813.7337;
   DATA[2289,14] := 1.0;
   DATA[2289,15] := 2.0;
   DATA[2289,16] := 1.0;
   DATA[2289,17] := 1.0;
   DATA[2289,18] := 1.0;
   DATA[2289,19] := 2.0;
   DATA[2289,20] := 148.808;
   DATA[2289,21] := 154.909;
   DATA[2289,22] := 1.720693;
   DATA[2289,23] := 850.705;
   DATA[2289,24] := 2.0;
   DATA[2289,25] := 2.0;
   DATA[2289,26] := 7.874455;
   DATA[2289,27] := 144.527;
   DATA[2289,28] := 261.7278;
   DATA[2289,29] := 11.95847;
   DATA[2289,30] := 1.730838;
   DATA[2289,31] := 1.291533;
   DATA[2289,32] := 0.7355248;
   DATA[2289,33] := 0.3083624;
   DATA[2289,34] := 2.0;
   DATA[2289,35] := 250.4005;
   DATA[2289,36] := 1.681991;
   DATA[2289,37] := 189.2944;
   DATA[2289,38] := 0.000128152;
   DATA[2289,39] := 1.0;
   DATA[2289,40] := 1.0;
   DATA[2290,0] := 2.533068;
   DATA[2290,1] := 864.8168;
   DATA[2290,2] := 2.0;
   DATA[2290,3] := 2.0;
   DATA[2290,4] := 262.3366;
   DATA[2290,5] := 8.395475;
   DATA[2290,6] := 330.0948;
   DATA[2290,7] := 2.455259;
   DATA[2290,8] := 2.0;
   DATA[2290,9] := 2.0;
   DATA[2290,10] := 2.0;
   DATA[2290,11] := 19.73238;
   DATA[2290,12] := 2.206963;
   DATA[2290,13] := 813.8138;
   DATA[2290,14] := 1.0;
   DATA[2290,15] := 2.0;
   DATA[2290,16] := 1.0;
   DATA[2290,17] := 1.0;
   DATA[2290,18] := 1.0;
   DATA[2290,19] := 2.0;
   DATA[2290,20] := 148.808;
   DATA[2290,21] := 154.909;
   DATA[2290,22] := 1.720693;
   DATA[2290,23] := 850.9741;
   DATA[2290,24] := 2.0;
   DATA[2290,25] := 2.0;
   DATA[2290,26] := 7.873174;
   DATA[2290,27] := 144.3989;
   DATA[2290,28] := 261.7278;
   DATA[2290,29] := 11.95847;
   DATA[2290,30] := 1.730069;
   DATA[2290,31] := 1.281927;
   DATA[2290,32] := 0.7355248;
   DATA[2290,33] := 0.3083624;
   DATA[2290,34] := 2.0;
   DATA[2290,35] := 250.4005;
   DATA[2290,36] := 1.681991;
   DATA[2290,37] := 189.2944;
   DATA[2290,38] := 0.000128152;
   DATA[2290,39] := 1.0;
   DATA[2290,40] := 1.0;
   DATA[2291,0] := 2.517695;
   DATA[2291,1] := 864.6597;
   DATA[2291,2] := 2.0;
   DATA[2291,3] := 2.0;
   DATA[2291,4] := 262.3366;
   DATA[2291,5] := 8.395475;
   DATA[2291,6] := 330.0948;
   DATA[2291,7] := 2.455259;
   DATA[2291,8] := 2.0;
   DATA[2291,9] := 2.0;
   DATA[2291,10] := 2.0;
   DATA[2291,11] := 19.73238;
   DATA[2291,12] := 2.206963;
   DATA[2291,13] := 814.3745;
   DATA[2291,14] := 1.0;
   DATA[2291,15] := 2.0;
   DATA[2291,16] := 1.0;
   DATA[2291,17] := 1.0;
   DATA[2291,18] := 1.0;
   DATA[2291,19] := 2.0;
   DATA[2291,20] := 148.808;
   DATA[2291,21] := 154.909;
   DATA[2291,22] := 1.720693;
   DATA[2291,23] := 851.0895;
   DATA[2291,24] := 2.0;
   DATA[2291,25] := 2.0;
   DATA[2291,26] := 7.873174;
   DATA[2291,27] := 144.3989;
   DATA[2291,28] := 261.7278;
   DATA[2291,29] := 11.95847;
   DATA[2291,30] := 1.726865;
   DATA[2291,31] := 1.281542;
   DATA[2291,32] := 0.7355248;
   DATA[2291,33] := 0.3083624;
   DATA[2291,34] := 2.0;
   DATA[2291,35] := 250.4005;
   DATA[2291,36] := 1.681991;
   DATA[2291,37] := 189.1022;
   DATA[2291,38] := 0.000128152;
   DATA[2291,39] := 1.0;
   DATA[2291,40] := 1.0;
   DATA[2292,0] := 2.504244;
   DATA[2292,1] := 864.9738;
   DATA[2292,2] := 2.0;
   DATA[2292,3] := 2.0;
   DATA[2292,4] := 262.3366;
   DATA[2292,5] := 8.395475;
   DATA[2292,6] := 330.0948;
   DATA[2292,7] := 2.455259;
   DATA[2292,8] := 2.0;
   DATA[2292,9] := 2.0;
   DATA[2292,10] := 2.0;
   DATA[2292,11] := 19.75479;
   DATA[2292,12] := 2.205169;
   DATA[2292,13] := 814.9353;
   DATA[2292,14] := 1.0;
   DATA[2292,15] := 2.0;
   DATA[2292,16] := 1.0;
   DATA[2292,17] := 1.0;
   DATA[2292,18] := 1.0;
   DATA[2292,19] := 2.0;
   DATA[2292,20] := 148.808;
   DATA[2292,21] := 154.909;
   DATA[2292,22] := 1.716464;
   DATA[2292,23] := 851.1664;
   DATA[2292,24] := 2.0;
   DATA[2292,25] := 2.0;
   DATA[2292,26] := 7.873174;
   DATA[2292,27] := 144.3989;
   DATA[2292,28] := 261.7278;
   DATA[2292,29] := 11.95847;
   DATA[2292,30] := 1.726352;
   DATA[2292,31] := 1.272576;
   DATA[2292,32] := 0.7348846;
   DATA[2292,33] := 0.3083624;
   DATA[2292,34] := 2.0;
   DATA[2292,35] := 250.4005;
   DATA[2292,36] := 1.681991;
   DATA[2292,37] := 189.1022;
   DATA[2292,38] := 0.000128152;
   DATA[2292,39] := 1.0;
   DATA[2292,40] := 1.0;
   DATA[2293,0] := 2.489511;
   DATA[2293,1] := 864.856;
   DATA[2293,2] := 2.0;
   DATA[2293,3] := 2.0;
   DATA[2293,4] := 262.3366;
   DATA[2293,5] := 8.395475;
   DATA[2293,6] := 330.0948;
   DATA[2293,7] := 2.455259;
   DATA[2293,8] := 2.0;
   DATA[2293,9] := 2.0;
   DATA[2293,10] := 2.0;
   DATA[2293,11] := 19.75479;
   DATA[2293,12] := 2.205169;
   DATA[2293,13] := 815.0154;
   DATA[2293,14] := 1.0;
   DATA[2293,15] := 2.0;
   DATA[2293,16] := 1.0;
   DATA[2293,17] := 1.0;
   DATA[2293,18] := 1.0;
   DATA[2293,19] := 2.0;
   DATA[2293,20] := 148.808;
   DATA[2293,21] := 154.909;
   DATA[2293,22] := 1.715567;
   DATA[2293,23] := 850.9741;
   DATA[2293,24] := 2.0;
   DATA[2293,25] := 2.0;
   DATA[2293,26] := 7.873174;
   DATA[2293,27] := 144.3989;
   DATA[2293,28] := 261.7278;
   DATA[2293,29] := 11.95847;
   DATA[2293,30] := 1.726352;
   DATA[2293,31] := 1.272576;
   DATA[2293,32] := 0.7348846;
   DATA[2293,33] := 0.3083624;
   DATA[2293,34] := 2.0;
   DATA[2293,35] := 250.1762;
   DATA[2293,36] := 1.681991;
   DATA[2293,37] := 189.1022;
   DATA[2293,38] := 0.000128152;
   DATA[2293,39] := 1.0;
   DATA[2293,40] := 1.0;
   DATA[2294,0] := 2.475419;
   DATA[2294,1] := 865.0523;
   DATA[2294,2] := 2.0;
   DATA[2294,3] := 2.0;
   DATA[2294,4] := 262.3366;
   DATA[2294,5] := 8.395475;
   DATA[2294,6] := 330.0948;
   DATA[2294,7] := 2.455259;
   DATA[2294,8] := 2.0;
   DATA[2294,9] := 2.0;
   DATA[2294,10] := 2.0;
   DATA[2294,11] := 19.70037;
   DATA[2294,12] := 2.205169;
   DATA[2294,13] := 815.5762;
   DATA[2294,14] := 1.0;
   DATA[2294,15] := 2.0;
   DATA[2294,16] := 1.0;
   DATA[2294,17] := 1.0;
   DATA[2294,18] := 1.0;
   DATA[2294,19] := 2.0;
   DATA[2294,20] := 148.808;
   DATA[2294,21] := 155.0115;
   DATA[2294,22] := 1.715567;
   DATA[2294,23] := 851.0895;
   DATA[2294,24] := 2.0;
   DATA[2294,25] := 2.0;
   DATA[2294,26] := 7.873174;
   DATA[2294,27] := 144.3989;
   DATA[2294,28] := 261.7278;
   DATA[2294,29] := 11.95847;
   DATA[2294,30] := 1.725583;
   DATA[2294,31] := 1.28103;
   DATA[2294,32] := 0.7348846;
   DATA[2294,33] := 0.3083624;
   DATA[2294,34] := 2.0;
   DATA[2294,35] := 250.1762;
   DATA[2294,36] := 1.681991;
   DATA[2294,37] := 189.1022;
   DATA[2294,38] := 0.000128152;
   DATA[2294,39] := 1.0;
   DATA[2294,40] := 1.0;
   DATA[2295,0] := 2.457803;
   DATA[2295,1] := 864.9345;
   DATA[2295,2] := 2.0;
   DATA[2295,3] := 2.0;
   DATA[2295,4] := 262.3366;
   DATA[2295,5] := 8.395475;
   DATA[2295,6] := 330.0948;
   DATA[2295,7] := 2.455259;
   DATA[2295,8] := 2.0;
   DATA[2295,9] := 2.0;
   DATA[2295,10] := 2.0;
   DATA[2295,11] := 19.70037;
   DATA[2295,12] := 2.205169;
   DATA[2295,13] := 815.3759;
   DATA[2295,14] := 1.0;
   DATA[2295,15] := 2.0;
   DATA[2295,16] := 1.0;
   DATA[2295,17] := 1.0;
   DATA[2295,18] := 1.0;
   DATA[2295,19] := 2.0;
   DATA[2295,20] := 148.808;
   DATA[2295,21] := 155.0115;
   DATA[2295,22] := 1.714926;
   DATA[2295,23] := 850.8203;
   DATA[2295,24] := 2.0;
   DATA[2295,25] := 2.0;
   DATA[2295,26] := 7.873174;
   DATA[2295,27] := 144.3989;
   DATA[2295,28] := 261.7278;
   DATA[2295,29] := 11.95847;
   DATA[2295,30] := 1.723148;
   DATA[2295,31] := 1.281798;
   DATA[2295,32] := 0.7348846;
   DATA[2295,33] := 0.3083624;
   DATA[2295,34] := 2.0;
   DATA[2295,35] := 250.1762;
   DATA[2295,36] := 1.681991;
   DATA[2295,37] := 189.1022;
   DATA[2295,38] := 0.000128152;
   DATA[2295,39] := 1.0;
   DATA[2295,40] := 1.0;
   DATA[2296,0] := 2.444992;
   DATA[2296,1] := 865.3663;
   DATA[2296,2] := 2.0;
   DATA[2296,3] := 2.0;
   DATA[2296,4] := 262.3366;
   DATA[2296,5] := 8.395475;
   DATA[2296,6] := 330.0948;
   DATA[2296,7] := 2.455259;
   DATA[2296,8] := 2.0;
   DATA[2296,9] := 2.0;
   DATA[2296,10] := 2.0;
   DATA[2296,11] := 19.70037;
   DATA[2296,12] := 2.203632;
   DATA[2296,13] := 815.7364;
   DATA[2296,14] := 1.0;
   DATA[2296,15] := 2.0;
   DATA[2296,16] := 1.0;
   DATA[2296,17] := 1.0;
   DATA[2296,18] := 1.0;
   DATA[2296,19] := 2.0;
   DATA[2296,20] := 148.808;
   DATA[2296,21] := 155.0115;
   DATA[2296,22] := 1.714926;
   DATA[2296,23] := 851.2817;
   DATA[2296,24] := 2.0;
   DATA[2296,25] := 2.0;
   DATA[2296,26] := 7.873174;
   DATA[2296,27] := 144.3989;
   DATA[2296,28] := 261.7278;
   DATA[2296,29] := 11.95847;
   DATA[2296,30] := 1.723148;
   DATA[2296,31] := 1.281798;
   DATA[2296,32] := 0.7348846;
   DATA[2296,33] := 0.3083624;
   DATA[2296,34] := 2.0;
   DATA[2296,35] := 250.1762;
   DATA[2296,36] := 1.681991;
   DATA[2296,37] := 188.958;
   DATA[2296,38] := 0.000128152;
   DATA[2296,39] := 1.0;
   DATA[2296,40] := 1.0;
   DATA[2297,0] := 2.431861;
   DATA[2297,1] := 865.1308;
   DATA[2297,2] := 2.0;
   DATA[2297,3] := 2.0;
   DATA[2297,4] := 262.3366;
   DATA[2297,5] := 8.395475;
   DATA[2297,6] := 330.0948;
   DATA[2297,7] := 2.455259;
   DATA[2297,8] := 2.0;
   DATA[2297,9] := 2.0;
   DATA[2297,10] := 2.0;
   DATA[2297,11] := 19.70037;
   DATA[2297,12] := 2.203632;
   DATA[2297,13] := 815.456;
   DATA[2297,14] := 1.0;
   DATA[2297,15] := 2.0;
   DATA[2297,16] := 1.0;
   DATA[2297,17] := 1.0;
   DATA[2297,18] := 1.0;
   DATA[2297,19] := 2.0;
   DATA[2297,20] := 148.808;
   DATA[2297,21] := 155.0115;
   DATA[2297,22] := 1.714926;
   DATA[2297,23] := 851.2433;
   DATA[2297,24] := 2.0;
   DATA[2297,25] := 2.0;
   DATA[2297,26] := 7.873174;
   DATA[2297,27] := 144.3989;
   DATA[2297,28] := 261.7278;
   DATA[2297,29] := 11.95847;
   DATA[2297,30] := 1.723148;
   DATA[2297,31] := 1.304214;
   DATA[2297,32] := 0.7348846;
   DATA[2297,33] := 0.3083624;
   DATA[2297,34] := 2.0;
   DATA[2297,35] := 250.1762;
   DATA[2297,36] := 1.681991;
   DATA[2297,37] := 188.958;
   DATA[2297,38] := 0.000128152;
   DATA[2297,39] := 1.0;
   DATA[2297,40] := 1.0;
   DATA[2298,0] := 2.425776;
   DATA[2298,1] := 865.4056;
   DATA[2298,2] := 2.0;
   DATA[2298,3] := 2.0;
   DATA[2298,4] := 262.3366;
   DATA[2298,5] := 8.395475;
   DATA[2298,6] := 330.0948;
   DATA[2298,7] := 2.455259;
   DATA[2298,8] := 2.0;
   DATA[2298,9] := 2.0;
   DATA[2298,10] := 2.0;
   DATA[2298,11] := 19.70037;
   DATA[2298,12] := 2.203632;
   DATA[2298,13] := 815.6162;
   DATA[2298,14] := 1.0;
   DATA[2298,15] := 2.0;
   DATA[2298,16] := 1.0;
   DATA[2298,17] := 1.0;
   DATA[2298,18] := 1.0;
   DATA[2298,19] := 2.0;
   DATA[2298,20] := 148.808;
   DATA[2298,21] := 155.0115;
   DATA[2298,22] := 1.714926;
   DATA[2298,23] := 851.3971;
   DATA[2298,24] := 2.0;
   DATA[2298,25] := 2.0;
   DATA[2298,26] := 7.873174;
   DATA[2298,27] := 144.3989;
   DATA[2298,28] := 261.7278;
   DATA[2298,29] := 11.95847;
   DATA[2298,30] := 1.723148;
   DATA[2298,31] := 1.310747;
   DATA[2298,32] := 0.7348846;
   DATA[2298,33] := 0.3083624;
   DATA[2298,34] := 2.0;
   DATA[2298,35] := 250.1762;
   DATA[2298,36] := 1.681991;
   DATA[2298,37] := 188.958;
   DATA[2298,38] := 0.000128152;
   DATA[2298,39] := 1.0;
   DATA[2298,40] := 1.0;
   DATA[2299,0] := 2.425456;
   DATA[2299,1] := 865.5626;
   DATA[2299,2] := 2.0;
   DATA[2299,3] := 2.0;
   DATA[2299,4] := 262.3366;
   DATA[2299,5] := 8.395475;
   DATA[2299,6] := 330.0948;
   DATA[2299,7] := 2.456156;
   DATA[2299,8] := 2.0;
   DATA[2299,9] := 2.0;
   DATA[2299,10] := 2.0;
   DATA[2299,11] := 19.67796;
   DATA[2299,12] := 2.206322;
   DATA[2299,13] := 815.416;
   DATA[2299,14] := 1.0;
   DATA[2299,15] := 2.0;
   DATA[2299,16] := 1.0;
   DATA[2299,17] := 1.0;
   DATA[2299,18] := 1.0;
   DATA[2299,19] := 2.0;
   DATA[2299,20] := 148.808;
   DATA[2299,21] := 155.0115;
   DATA[2299,22] := 1.714926;
   DATA[2299,23] := 851.3971;
   DATA[2299,24] := 2.0;
   DATA[2299,25] := 2.0;
   DATA[2299,26] := 7.874776;
   DATA[2299,27] := 144.5014;
   DATA[2299,28] := 261.7278;
   DATA[2299,29] := 11.95847;
   DATA[2299,30] := 1.725327;
   DATA[2299,31] := 1.311772;
   DATA[2299,32] := 0.7348846;
   DATA[2299,33] := 0.3083624;
   DATA[2299,34] := 2.0;
   DATA[2299,35] := 250.1762;
   DATA[2299,36] := 1.681991;
   DATA[2299,37] := 188.958;
   DATA[2299,38] := 0.000128152;
   DATA[2299,39] := 1.0;
   DATA[2299,40] := 1.0;
   DATA[2300,0] := 2.451398;
   DATA[2300,1] := 865.7589;
   DATA[2300,2] := 2.0;
   DATA[2300,3] := 2.0;
   DATA[2300,4] := 262.3366;
   DATA[2300,5] := 8.395475;
   DATA[2300,6] := 330.0948;
   DATA[2300,7] := 2.456156;
   DATA[2300,8] := 2.0;
   DATA[2300,9] := 2.0;
   DATA[2300,10] := 2.0;
   DATA[2300,11] := 19.65235;
   DATA[2300,12] := 2.207091;
   DATA[2300,13] := 815.2157;
   DATA[2300,14] := 1.0;
   DATA[2300,15] := 2.0;
   DATA[2300,16] := 1.0;
   DATA[2300,17] := 1.0;
   DATA[2300,18] := 1.0;
   DATA[2300,19] := 2.0;
   DATA[2300,20] := 148.808;
   DATA[2300,21] := 155.0115;
   DATA[2300,22] := 1.717874;
   DATA[2300,23] := 851.7432;
   DATA[2300,24] := 2.0;
   DATA[2300,25] := 2.0;
   DATA[2300,26] := 7.874776;
   DATA[2300,27] := 144.5014;
   DATA[2300,28] := 261.7278;
   DATA[2300,29] := 11.95847;
   DATA[2300,30] := 1.725327;
   DATA[2300,31] := 1.312284;
   DATA[2300,32] := 0.7348846;
   DATA[2300,33] := 0.3083624;
   DATA[2300,34] := 2.0;
   DATA[2300,35] := 250.1762;
   DATA[2300,36] := 1.681991;
   DATA[2300,37] := 188.958;
   DATA[2300,38] := 0.000128152;
   DATA[2300,39] := 1.0;
   DATA[2300,40] := 1.0;
   DATA[2301,0] := 2.498479;
   DATA[2301,1] := 865.7981;
   DATA[2301,2] := 2.0;
   DATA[2301,3] := 2.0;
   DATA[2301,4] := 262.3366;
   DATA[2301,5] := 8.395475;
   DATA[2301,6] := 330.0948;
   DATA[2301,7] := 2.456156;
   DATA[2301,8] := 2.0;
   DATA[2301,9] := 2.0;
   DATA[2301,10] := 2.0;
   DATA[2301,11] := 19.65235;
   DATA[2301,12] := 2.207091;
   DATA[2301,13] := 814.8552;
   DATA[2301,14] := 1.0;
   DATA[2301,15] := 2.0;
   DATA[2301,16] := 1.0;
   DATA[2301,17] := 1.0;
   DATA[2301,18] := 1.0;
   DATA[2301,19] := 2.0;
   DATA[2301,20] := 148.808;
   DATA[2301,21] := 155.0884;
   DATA[2301,22] := 1.718515;
   DATA[2301,23] := 851.3971;
   DATA[2301,24] := 2.0;
   DATA[2301,25] := 2.0;
   DATA[2301,26] := 7.874776;
   DATA[2301,27] := 144.5014;
   DATA[2301,28] := 261.7278;
   DATA[2301,29] := 11.95847;
   DATA[2301,30] := 1.725711;
   DATA[2301,31] := 1.298578;
   DATA[2301,32] := 0.7353967;
   DATA[2301,33] := 0.3083624;
   DATA[2301,34] := 2.0;
   DATA[2301,35] := 250.1762;
   DATA[2301,36] := 1.681991;
   DATA[2301,37] := 188.958;
   DATA[2301,38] := 0.000128152;
   DATA[2301,39] := 1.0;
   DATA[2301,40] := 1.0;
   DATA[2302,0] := 2.539474;
   DATA[2302,1] := 866.1906;
   DATA[2302,2] := 2.0;
   DATA[2302,3] := 2.0;
   DATA[2302,4] := 262.3366;
   DATA[2302,5] := 8.395475;
   DATA[2302,6] := 330.0948;
   DATA[2302,7] := 2.456156;
   DATA[2302,8] := 2.0;
   DATA[2302,9] := 2.0;
   DATA[2302,10] := 2.0;
   DATA[2302,11] := 19.69396;
   DATA[2302,12] := 2.207091;
   DATA[2302,13] := 814.8552;
   DATA[2302,14] := 1.0;
   DATA[2302,15] := 2.0;
   DATA[2302,16] := 1.0;
   DATA[2302,17] := 1.0;
   DATA[2302,18] := 1.0;
   DATA[2302,19] := 2.0;
   DATA[2302,20] := 148.808;
   DATA[2302,21] := 155.0884;
   DATA[2302,22] := 1.718515;
   DATA[2302,23] := 851.3971;
   DATA[2302,24] := 2.0;
   DATA[2302,25] := 2.0;
   DATA[2302,26] := 7.874776;
   DATA[2302,27] := 144.5014;
   DATA[2302,28] := 261.7278;
   DATA[2302,29] := 11.95847;
   DATA[2302,30] := 1.727634;
   DATA[2302,31] := 1.292046;
   DATA[2302,32] := 0.7353967;
   DATA[2302,33] := 0.3083624;
   DATA[2302,34] := 2.0;
   DATA[2302,35] := 250.1762;
   DATA[2302,36] := 1.681991;
   DATA[2302,37] := 189.1022;
   DATA[2302,38] := 0.000128152;
   DATA[2302,39] := 1.0;
   DATA[2302,40] := 1.0;
   DATA[2303,0] := 2.580149;
   DATA[2303,1] := 865.7981;
   DATA[2303,2] := 2.0;
   DATA[2303,3] := 2.0;
   DATA[2303,4] := 262.3366;
   DATA[2303,5] := 8.395475;
   DATA[2303,6] := 330.0948;
   DATA[2303,7] := 2.457566;
   DATA[2303,8] := 2.0;
   DATA[2303,9] := 2.0;
   DATA[2303,10] := 2.0;
   DATA[2303,11] := 19.69396;
   DATA[2303,12] := 2.207091;
   DATA[2303,13] := 814.7751;
   DATA[2303,14] := 1.0;
   DATA[2303,15] := 2.0;
   DATA[2303,16] := 1.0;
   DATA[2303,17] := 1.0;
   DATA[2303,18] := 1.0;
   DATA[2303,19] := 2.0;
   DATA[2303,20] := 148.808;
   DATA[2303,21] := 155.0884;
   DATA[2303,22] := 1.718515;
   DATA[2303,23] := 852.0508;
   DATA[2303,24] := 2.0;
   DATA[2303,25] := 2.0;
   DATA[2303,26] := 7.874776;
   DATA[2303,27] := 144.5014;
   DATA[2303,28] := 261.7278;
   DATA[2303,29] := 11.95847;
   DATA[2303,30] := 1.727634;
   DATA[2303,31] := 1.300884;
   DATA[2303,32] := 0.7353967;
   DATA[2303,33] := 0.3083624;
   DATA[2303,34] := 2.0;
   DATA[2303,35] := 250.1762;
   DATA[2303,36] := 1.681991;
   DATA[2303,37] := 189.1662;
   DATA[2303,38] := 0.000128152;
   DATA[2303,39] := 1.0;
   DATA[2303,40] := 1.0;
   DATA[2304,0] := 2.620824;
   DATA[2304,1] := 865.9551;
   DATA[2304,2] := 2.0;
   DATA[2304,3] := 2.0;
   DATA[2304,4] := 262.3366;
   DATA[2304,5] := 8.395475;
   DATA[2304,6] := 330.0948;
   DATA[2304,7] := 2.457566;
   DATA[2304,8] := 2.0;
   DATA[2304,9] := 2.0;
   DATA[2304,10] := 2.0;
   DATA[2304,11] := 19.69396;
   DATA[2304,12] := 2.207091;
   DATA[2304,13] := 814.8151;
   DATA[2304,14] := 1.0;
   DATA[2304,15] := 2.0;
   DATA[2304,16] := 1.0;
   DATA[2304,17] := 1.0;
   DATA[2304,18] := 1.0;
   DATA[2304,19] := 2.0;
   DATA[2304,20] := 148.808;
   DATA[2304,21] := 155.0884;
   DATA[2304,22] := 1.718515;
   DATA[2304,23] := 852.4353;
   DATA[2304,24] := 2.0;
   DATA[2304,25] := 2.0;
   DATA[2304,26] := 7.874776;
   DATA[2304,27] := 144.5014;
   DATA[2304,28] := 261.7278;
   DATA[2304,29] := 11.95847;
   DATA[2304,30] := 1.727634;
   DATA[2304,31] := 1.305367;
   DATA[2304,32] := 0.7353967;
   DATA[2304,33] := 0.3083624;
   DATA[2304,34] := 2.0;
   DATA[2304,35] := 250.3044;
   DATA[2304,36] := 1.681991;
   DATA[2304,37] := 189.1662;
   DATA[2304,38] := 0.000128152;
   DATA[2304,39] := 1.0;
   DATA[2304,40] := 1.0;
   DATA[2305,0] := 2.641642;
   DATA[2305,1] := 865.9551;
   DATA[2305,2] := 2.0;
   DATA[2305,3] := 2.0;
   DATA[2305,4] := 262.3366;
   DATA[2305,5] := 8.395475;
   DATA[2305,6] := 330.0436;
   DATA[2305,7] := 2.457566;
   DATA[2305,8] := 2.0;
   DATA[2305,9] := 2.0;
   DATA[2305,10] := 2.0;
   DATA[2305,11] := 19.69396;
   DATA[2305,12] := 2.208372;
   DATA[2305,13] := 814.735;
   DATA[2305,14] := 1.0;
   DATA[2305,15] := 2.0;
   DATA[2305,16] := 1.0;
   DATA[2305,17] := 1.0;
   DATA[2305,18] := 1.0;
   DATA[2305,19] := 2.0;
   DATA[2305,20] := 148.808;
   DATA[2305,21] := 155.0884;
   DATA[2305,22] := 1.718515;
   DATA[2305,23] := 852.5506;
   DATA[2305,24] := 2.0;
   DATA[2305,25] := 2.0;
   DATA[2305,26] := 7.874455;
   DATA[2305,27] := 144.5014;
   DATA[2305,28] := 261.7278;
   DATA[2305,29] := 11.95847;
   DATA[2305,30] := 1.725455;
   DATA[2305,31] := 1.311003;
   DATA[2305,32] := 0.7353967;
   DATA[2305,33] := 0.3083624;
   DATA[2305,34] := 2.0;
   DATA[2305,35] := 250.3525;
   DATA[2305,36] := 1.681991;
   DATA[2305,37] := 189.1662;
   DATA[2305,38] := 0.000128152;
   DATA[2305,39] := 1.0;
   DATA[2305,40] := 1.0;
   DATA[2306,0] := 2.657016;
   DATA[2306,1] := 866.2691;
   DATA[2306,2] := 2.0;
   DATA[2306,3] := 2.0;
   DATA[2306,4] := 262.3366;
   DATA[2306,5] := 8.395475;
   DATA[2306,6] := 329.9667;
   DATA[2306,7] := 2.457566;
   DATA[2306,8] := 2.0;
   DATA[2306,9] := 2.0;
   DATA[2306,10] := 2.0;
   DATA[2306,11] := 19.69396;
   DATA[2306,12] := 2.208884;
   DATA[2306,13] := 815.0154;
   DATA[2306,14] := 1.0;
   DATA[2306,15] := 2.0;
   DATA[2306,16] := 1.0;
   DATA[2306,17] := 1.0;
   DATA[2306,18] := 1.0;
   DATA[2306,19] := 2.0;
   DATA[2306,20] := 148.808;
   DATA[2306,21] := 155.0884;
   DATA[2306,22] := 1.718515;
   DATA[2306,23] := 853.1274;
   DATA[2306,24] := 2.0;
   DATA[2306,25] := 2.0;
   DATA[2306,26] := 7.874455;
   DATA[2306,27] := 144.5014;
   DATA[2306,28] := 261.5355;
   DATA[2306,29] := 11.95847;
   DATA[2306,30] := 1.725455;
   DATA[2306,31] := 1.312284;
   DATA[2306,32] := 0.7353967;
   DATA[2306,33] := 0.3083624;
   DATA[2306,34] := 2.0;
   DATA[2306,35] := 250.3525;
   DATA[2306,36] := 1.681991;
   DATA[2306,37] := 189.1662;
   DATA[2306,38] := 0.000128152;
   DATA[2306,39] := 1.0;
   DATA[2306,40] := 1.0;
   DATA[2307,0] := 2.657336;
   DATA[2307,1] := 866.3083;
   DATA[2307,2] := 2.0;
   DATA[2307,3] := 2.0;
   DATA[2307,4] := 262.3366;
   DATA[2307,5] := 8.395475;
   DATA[2307,6] := 329.9667;
   DATA[2307,7] := 2.456541;
   DATA[2307,8] := 2.0;
   DATA[2307,9] := 2.0;
   DATA[2307,10] := 2.0;
   DATA[2307,11] := 19.69396;
   DATA[2307,12] := 2.208884;
   DATA[2307,13] := 814.4547;
   DATA[2307,14] := 1.0;
   DATA[2307,15] := 2.0;
   DATA[2307,16] := 1.0;
   DATA[2307,17] := 1.0;
   DATA[2307,18] := 1.0;
   DATA[2307,19] := 2.0;
   DATA[2307,20] := 148.808;
   DATA[2307,21] := 155.0884;
   DATA[2307,22] := 1.718515;
   DATA[2307,23] := 853.5119;
   DATA[2307,24] := 2.0;
   DATA[2307,25] := 2.0;
   DATA[2307,26] := 7.874455;
   DATA[2307,27] := 144.5014;
   DATA[2307,28] := 261.5355;
   DATA[2307,29] := 11.95847;
   DATA[2307,30] := 1.725455;
   DATA[2307,31] := 1.301012;
   DATA[2307,32] := 0.7353967;
   DATA[2307,33] := 0.3083624;
   DATA[2307,34] := 2.0;
   DATA[2307,35] := 250.3525;
   DATA[2307,36] := 1.681991;
   DATA[2307,37] := 189.1662;
   DATA[2307,38] := 0.000128152;
   DATA[2307,39] := 1.0;
   DATA[2307,40] := 1.0;
   DATA[2308,0] := 2.639721;
   DATA[2308,1] := 866.4654;
   DATA[2308,2] := 2.0;
   DATA[2308,3] := 2.0;
   DATA[2308,4] := 262.3366;
   DATA[2308,5] := 8.395475;
   DATA[2308,6] := 329.9667;
   DATA[2308,7] := 2.456541;
   DATA[2308,8] := 2.0;
   DATA[2308,9] := 2.0;
   DATA[2308,10] := 2.0;
   DATA[2308,11] := 19.69396;
   DATA[2308,12] := 2.208884;
   DATA[2308,13] := 814.735;
   DATA[2308,14] := 1.0;
   DATA[2308,15] := 2.0;
   DATA[2308,16] := 1.0;
   DATA[2308,17] := 1.0;
   DATA[2308,18] := 1.0;
   DATA[2308,19] := 2.0;
   DATA[2308,20] := 148.808;
   DATA[2308,21] := 155.0884;
   DATA[2308,22] := 1.717746;
   DATA[2308,23] := 853.3965;
   DATA[2308,24] := 2.0;
   DATA[2308,25] := 2.0;
   DATA[2308,26] := 7.874135;
   DATA[2308,27] := 144.5014;
   DATA[2308,28] := 261.5355;
   DATA[2308,29] := 11.95847;
   DATA[2308,30] := 1.725455;
   DATA[2308,31] := 1.29243;
   DATA[2308,32] := 0.7353967;
   DATA[2308,33] := 0.3083624;
   DATA[2308,34] := 2.0;
   DATA[2308,35] := 250.3525;
   DATA[2308,36] := 1.681991;
   DATA[2308,37] := 189.1662;
   DATA[2308,38] := 0.000128152;
   DATA[2308,39] := 1.0;
   DATA[2308,40] := 1.0;
   DATA[2309,0] := 2.624347;
   DATA[2309,1] := 866.1906;
   DATA[2309,2] := 2.0;
   DATA[2309,3] := 2.0;
   DATA[2309,4] := 262.3366;
   DATA[2309,5] := 8.395475;
   DATA[2309,6] := 329.9667;
   DATA[2309,7] := 2.456541;
   DATA[2309,8] := 2.0;
   DATA[2309,9] := 2.0;
   DATA[2309,10] := 2.0;
   DATA[2309,11] := 19.72598;
   DATA[2309,12] := 2.209653;
   DATA[2309,13] := 814.2143;
   DATA[2309,14] := 1.0;
   DATA[2309,15] := 2.0;
   DATA[2309,16] := 1.0;
   DATA[2309,17] := 1.0;
   DATA[2309,18] := 1.0;
   DATA[2309,19] := 2.0;
   DATA[2309,20] := 148.808;
   DATA[2309,21] := 155.0884;
   DATA[2309,22] := 1.71608;
   DATA[2309,23] := 853.858;
   DATA[2309,24] := 2.0;
   DATA[2309,25] := 2.0;
   DATA[2309,26] := 7.874135;
   DATA[2309,27] := 144.5014;
   DATA[2309,28] := 261.5355;
   DATA[2309,29] := 11.95847;
   DATA[2309,30] := 1.725455;
   DATA[2309,31] := 1.292174;
   DATA[2309,32] := 0.7353967;
   DATA[2309,33] := 0.3083624;
   DATA[2309,34] := 2.0;
   DATA[2309,35] := 250.2403;
   DATA[2309,36] := 1.681991;
   DATA[2309,37] := 189.0381;
   DATA[2309,38] := 0.000128152;
   DATA[2309,39] := 1.0;
   DATA[2309,40] := 1.0;
   DATA[2310,0] := 2.618582;
   DATA[2310,1] := 866.5831;
   DATA[2310,2] := 2.0;
   DATA[2310,3] := 2.0;
   DATA[2310,4] := 262.3366;
   DATA[2310,5] := 8.395475;
   DATA[2310,6] := 329.9667;
   DATA[2310,7] := 2.456541;
   DATA[2310,8] := 2.0;
   DATA[2310,9] := 2.0;
   DATA[2310,10] := 2.0;
   DATA[2310,11] := 19.73238;
   DATA[2310,12] := 2.210166;
   DATA[2310,13] := 814.6149;
   DATA[2310,14] := 1.0;
   DATA[2310,15] := 2.0;
   DATA[2310,16] := 1.0;
   DATA[2310,17] := 1.0;
   DATA[2310,18] := 1.0;
   DATA[2310,19] := 2.0;
   DATA[2310,20] := 148.808;
   DATA[2310,21] := 155.0884;
   DATA[2310,22] := 1.715952;
   DATA[2310,23] := 853.7811;
   DATA[2310,24] := 2.0;
   DATA[2310,25] := 2.0;
   DATA[2310,26] := 7.874135;
   DATA[2310,27] := 144.5014;
   DATA[2310,28] := 261.5355;
   DATA[2310,29] := 11.95847;
   DATA[2310,30] := 1.725455;
   DATA[2310,31] := 1.292174;
   DATA[2310,32] := 0.7353967;
   DATA[2310,33] := 0.3083624;
   DATA[2310,34] := 2.0;
   DATA[2310,35] := 250.2403;
   DATA[2310,36] := 1.681991;
   DATA[2310,37] := 189.0381;
   DATA[2310,38] := 0.000128152;
   DATA[2310,39] := 1.0;
   DATA[2310,40] := 1.0;
   DATA[2311,0] := 2.612818;
   DATA[2311,1] := 866.1121;
   DATA[2311,2] := 2.0;
   DATA[2311,3] := 2.0;
   DATA[2311,4] := 262.3366;
   DATA[2311,5] := 8.395475;
   DATA[2311,6] := 329.9667;
   DATA[2311,7] := 2.456541;
   DATA[2311,8] := 2.0;
   DATA[2311,9] := 2.0;
   DATA[2311,10] := 2.0;
   DATA[2311,11] := 19.66835;
   DATA[2311,12] := 2.210166;
   DATA[2311,13] := 814.4547;
   DATA[2311,14] := 1.0;
   DATA[2311,15] := 2.0;
   DATA[2311,16] := 1.0;
   DATA[2311,17] := 1.0;
   DATA[2311,18] := 1.0;
   DATA[2311,19] := 2.0;
   DATA[2311,20] := 148.808;
   DATA[2311,21] := 155.0884;
   DATA[2311,22] := 1.715952;
   DATA[2311,23] := 854.1271;
   DATA[2311,24] := 2.0;
   DATA[2311,25] := 2.0;
   DATA[2311,26] := 7.874135;
   DATA[2311,27] := 144.5014;
   DATA[2311,28] := 261.5996;
   DATA[2311,29] := 11.95847;
   DATA[2311,30] := 1.725455;
   DATA[2311,31] := 1.292174;
   DATA[2311,32] := 0.7353967;
   DATA[2311,33] := 0.3083624;
   DATA[2311,34] := 2.0;
   DATA[2311,35] := 250.2403;
   DATA[2311,36] := 1.681991;
   DATA[2311,37] := 189.0381;
   DATA[2311,38] := 0.000128152;
   DATA[2311,39] := 1.0;
   DATA[2311,40] := 1.0;
   DATA[2312,0] := 2.598405;
   DATA[2312,1] := 865.6803;
   DATA[2312,2] := 2.0;
   DATA[2312,3] := 2.0;
   DATA[2312,4] := 262.3366;
   DATA[2312,5] := 8.395475;
   DATA[2312,6] := 329.9667;
   DATA[2312,7] := 2.456541;
   DATA[2312,8] := 2.0;
   DATA[2312,9] := 2.0;
   DATA[2312,10] := 2.0;
   DATA[2312,11] := 19.62994;
   DATA[2312,12] := 2.210166;
   DATA[2312,13] := 814.7751;
   DATA[2312,14] := 1.0;
   DATA[2312,15] := 2.0;
   DATA[2312,16] := 1.0;
   DATA[2312,17] := 1.0;
   DATA[2312,18] := 1.0;
   DATA[2312,19] := 2.0;
   DATA[2312,20] := 148.808;
   DATA[2312,21] := 155.0884;
   DATA[2312,22] := 1.715952;
   DATA[2312,23] := 854.2425;
   DATA[2312,24] := 2.0;
   DATA[2312,25] := 2.0;
   DATA[2312,26] := 7.874135;
   DATA[2312,27] := 144.5014;
   DATA[2312,28] := 261.8239;
   DATA[2312,29] := 11.95847;
   DATA[2312,30] := 1.725455;
   DATA[2312,31] := 1.300115;
   DATA[2312,32] := 0.7353967;
   DATA[2312,33] := 0.3083624;
   DATA[2312,34] := 2.0;
   DATA[2312,35] := 250.2403;
   DATA[2312,36] := 1.681991;
   DATA[2312,37] := 189.0381;
   DATA[2312,38] := 0.000128152;
   DATA[2312,39] := 1.0;
   DATA[2312,40] := 1.0;
   DATA[2313,0] := 2.582071;
   DATA[2313,1] := 865.6803;
   DATA[2313,2] := 2.0;
   DATA[2313,3] := 2.0;
   DATA[2313,4] := 262.3366;
   DATA[2313,5] := 8.395475;
   DATA[2313,6] := 330.1718;
   DATA[2313,7] := 2.456541;
   DATA[2313,8] := 2.0;
   DATA[2313,9] := 2.0;
   DATA[2313,10] := 2.0;
   DATA[2313,11] := 19.62994;
   DATA[2313,12] := 2.210166;
   DATA[2313,13] := 814.6149;
   DATA[2313,14] := 1.0;
   DATA[2313,15] := 2.0;
   DATA[2313,16] := 1.0;
   DATA[2313,17] := 1.0;
   DATA[2313,18] := 1.0;
   DATA[2313,19] := 2.0;
   DATA[2313,20] := 148.808;
   DATA[2313,21] := 155.0884;
   DATA[2313,22] := 1.715952;
   DATA[2313,23] := 854.4732;
   DATA[2313,24] := 2.0;
   DATA[2313,25] := 2.0;
   DATA[2313,26] := 7.874135;
   DATA[2313,27] := 144.5014;
   DATA[2313,28] := 261.8239;
   DATA[2313,29] := 11.95847;
   DATA[2313,30] := 1.725455;
   DATA[2313,31] := 1.297041;
   DATA[2313,32] := 0.7353967;
   DATA[2313,33] := 0.3083624;
   DATA[2313,34] := 2.0;
   DATA[2313,35] := 250.1122;
   DATA[2313,36] := 1.681991;
   DATA[2313,37] := 189.0381;
   DATA[2313,38] := 0.000128152;
   DATA[2313,39] := 1.0;
   DATA[2313,40] := 1.0;
   DATA[2314,0] := 2.564456;
   DATA[2314,1] := 865.7981;
   DATA[2314,2] := 2.0;
   DATA[2314,3] := 2.0;
   DATA[2314,4] := 262.3366;
   DATA[2314,5] := 8.395475;
   DATA[2314,6] := 330.1718;
   DATA[2314,7] := 2.456541;
   DATA[2314,8] := 2.0;
   DATA[2314,9] := 2.0;
   DATA[2314,10] := 2.0;
   DATA[2314,11] := 19.62994;
   DATA[2314,12] := 2.210166;
   DATA[2314,13] := 814.9353;
   DATA[2314,14] := 1.0;
   DATA[2314,15] := 2.0;
   DATA[2314,16] := 1.0;
   DATA[2314,17] := 1.0;
   DATA[2314,18] := 1.0;
   DATA[2314,19] := 2.0;
   DATA[2314,20] := 148.808;
   DATA[2314,21] := 155.0884;
   DATA[2314,22] := 1.715952;
   DATA[2314,23] := 854.5501;
